gfCNCPoint4[15652] = {X 437.5566, Y 8.7395, Z -5.5000, A 0.000, B 0.000, C 0.000 }
gfCNCPoint4[15653] = {X 439.1460, Y 8.3375, Z -5.5000, A 0.000, B 0.000, C 0.000 }
gfCNCPoint4[15654] = {X 441.2360, Y 8.0482, Z -5.5000, A 0.000, B 0.000, C 0.000 }
gfCNCPoint4[15655] = {X 443.3437, Y 7.9543, Z -5.5000, A 0.000, B 0.000, C 0.000 }
gfCNCPoint4[15656] = {X 444.0360, Y 7.9502, Z -5.5000, A 0.000, B 0.000, C 0.000 }
gfCNCPoint4[15657] = {X 459.4468, Y 7.9502, Z -5.5000, A 0.000, B 0.000, C 0.000 }
gfCNCPoint4[15658] = {X 460.3883, Y 8.0563, Z -5.5000, A 0.000, B 0.000, C 0.000 }
gfCNCPoint4[15659] = {X 461.2826, Y 8.3693, Z -5.5000, A 0.000, B 0.000, C 0.000 }
gfCNCPoint4[15660] = {X 462.0849, Y 8.8733, Z -5.5000, A 0.000, B 0.000, C 0.000 }
gfCNCPoint4[15661] = {X 462.7548, Y 9.5433, Z -5.5000, A 0.000, B 0.000, C 0.000 }
gfCNCPoint4[15662] = {X 463.2589, Y 10.3456, Z -5.5000, A 0.000, B 0.000, C 0.000 }
gfCNCPoint4[15663] = {X 463.5719, Y 11.2399, Z -5.5000, A 0.000, B 0.000, C 0.000 }
gfCNCPoint4[15664] = {X 463.6779, Y 12.1814, Z -5.5000, A 0.000, B 0.000, C 0.000 }
gfCNCPoint4[15665] = {X 463.6779, Y 12.9782, Z -5.5000, A 0.000, B 0.000, C 0.000 }
gfCNCPoint4[15666] = {X 463.5765, Y 13.8997, Z -5.5000, A 0.000, B 0.000, C 0.000 }
gfCNCPoint4[15667] = {X 463.2771, Y 14.7771, Z -5.5000, A 0.000, B 0.000, C 0.000 }
gfCNCPoint4[15668] = {X 462.7943, Y 15.5685, Z -5.5000, A 0.000, B 0.000, C 0.000 }
gfCNCPoint4[15669] = {X 462.1509, Y 16.2360, Z -5.5000, A 0.000, B 0.000, C 0.000 }
gfCNCPoint4[15670] = {X 462.1511, Y 28.5935, Z -5.5000, A 0.000, B 0.000, C 0.000 }
gfCNCPoint4[15671] = {X 466.1511, Y 28.5934, Z -5.5000, A 0.000, B 0.000, C 0.000 }
gfCNCPoint4[15672] = {X 462.0711, Y 28.5935, Z -5.5000, A 0.000, B 0.000, C 0.000 }
gfCNCPoint4[15673] = {X 462.0714, Y 40.9895, Z -5.5000, A 0.000, B 0.000, C 0.000 }
gfCNCPoint4[15674] = {X 462.1372, Y 41.0434, Z -5.5000, A 0.000, B 0.000, C 0.000 }
gfCNCPoint4[15675] = {X 462.7480, Y 41.6890, Z -5.5000, A 0.000, B 0.000, C 0.000 }
gfCNCPoint4[15676] = {X 463.2076, Y 42.4496, Z -5.5000, A 0.000, B 0.000, C 0.000 }
gfCNCPoint4[15677] = {X 463.4953, Y 43.2904, Z -5.5000, A 0.000, B 0.000, C 0.000 }
gfCNCPoint4[15678] = {X 463.5978, Y 44.1731, Z -5.5000, A 0.000, B 0.000, C 0.000 }
gfCNCPoint4[15679] = {X 463.5979, Y 45.0000, Z -5.5000, A 0.000, B 0.000, C 0.000 }
gfCNCPoint4[15680] = {X 463.4936, Y 45.9257, Z -5.5000, A 0.000, B 0.000, C 0.000 }
gfCNCPoint4[15681] = {X 463.1860, Y 46.8050, Z -5.5000, A 0.000, B 0.000, C 0.000 }
gfCNCPoint4[15682] = {X 462.6904, Y 47.5937, Z -5.5000, A 0.000, B 0.000, C 0.000 }
gfCNCPoint4[15683] = {X 462.0317, Y 48.2524, Z -5.5000, A 0.000, B 0.000, C 0.000 }
gfCNCPoint4[15684] = {X 461.2429, Y 48.7480, Z -5.5000, A 0.000, B 0.000, C 0.000 }
gfCNCPoint4[15685] = {X 460.3636, Y 49.0557, Z -5.5000, A 0.000, B 0.000, C 0.000 }
gfCNCPoint4[15686] = {X 459.4379, Y 49.1600, Z -5.5000, A 0.000, B 0.000, C 0.000 }
gfCNCPoint4[15687] = {X 452.9945, Y 49.1600, Z -5.5000, A 0.000, B 0.000, C 0.000 }
gfCNCPoint4[15688] = {X 452.0735, Y 49.0568, Z -5.5000, A 0.000, B 0.000, C 0.000 }
gfCNCPoint4[15689] = {X 451.1982, Y 48.7522, Z -5.5000, A 0.000, B 0.000, C 0.000 }
gfCNCPoint4[15690] = {X 450.4120, Y 48.2614, Z -5.5000, A 0.000, B 0.000, C 0.000 }
gfCNCPoint4[15691] = {X 449.7541, Y 47.6087, Z -5.5000, A 0.000, B 0.000, C 0.000 }
gfCNCPoint4[15692] = {X 449.2569, Y 46.8266, Z -5.5000, A 0.000, B 0.000, C 0.000 }
gfCNCPoint4[15693] = {X 448.9453, Y 45.9538, Z -5.5000, A 0.000, B 0.000, C 0.000 }
gfCNCPoint4[15694] = {X 448.8346, Y 45.0336, Z -5.5000, A 0.000, B 0.000, C 0.000 }
gfCNCPoint4[15695] = {X 448.8349, Y 44.1516, Z -5.5000, A 0.000, B 0.000, C 0.000 }
gfCNCPoint4[15696] = {X 448.9454, Y 43.2545, Z -5.5000, A 0.000, B 0.000, C 0.000 }
gfCNCPoint4[15697] = {X 449.2471, Y 42.4026, Z -5.5000, A 0.000, B 0.000, C 0.000 }
gfCNCPoint4[15698] = {X 449.7256, Y 41.6358, Z -5.5000, A 0.000, B 0.000, C 0.000 }
gfCNCPoint4[15699] = {X 450.3584, Y 40.9906, Z -5.5000, A 0.000, B 0.000, C 0.000 }
gfCNCPoint4[15700] = {X 450.3584, Y 34.3138, Z -5.5000, A 0.000, B 0.000, C 0.000 }
gfCNCPoint4[15701] = {X 447.3773, Y 34.3138, Z -5.5000, A 0.000, B 0.000, C 0.000 }
gfCNCPoint4[15702] = {X 443.0156, Y 42.8061, Z -5.5000, A 0.000, B 0.000, C 0.000 }
gfCNCPoint4[15703] = {X 443.0437, Y 42.8834, Z -5.5000, A 0.000, B 0.000, C 0.000 }
gfCNCPoint4[15704] = {X 443.2029, Y 43.5190, Z -5.5000, A 0.000, B 0.000, C 0.000 }
gfCNCPoint4[15705] = {X 443.2603, Y 44.1717, Z -5.5000, A 0.000, B 0.000, C 0.000 }
gfCNCPoint4[15706] = {X 443.2605, Y 45.0000, Z -5.5000, A 0.000, B 0.000, C 0.000 }
gfCNCPoint4[15707] = {X 443.1562, Y 45.9257, Z -5.5000, A 0.000, B 0.000, C 0.000 }
gfCNCPoint4[15708] = {X 442.8485, Y 46.8050, Z -5.5000, A 0.000, B 0.000, C 0.000 }
gfCNCPoint4[15709] = {X 442.3529, Y 47.5937, Z -5.5000, A 0.000, B 0.000, C 0.000 }
gfCNCPoint4[15710] = {X 441.6942, Y 48.2524, Z -5.5000, A 0.000, B 0.000, C 0.000 }
gfCNCPoint4[15711] = {X 440.9054, Y 48.7480, Z -5.5000, A 0.000, B 0.000, C 0.000 }
gfCNCPoint4[15712] = {X 440.0262, Y 49.0557, Z -5.5000, A 0.000, B 0.000, C 0.000 }
gfCNCPoint4[15713] = {X 439.1005, Y 49.1600, Z -5.5000, A 0.000, B 0.000, C 0.000 }
gfCNCPoint4[15714] = {X 432.5144, Y 49.1600, Z -5.5000, A 0.000, B 0.000, C 0.000 }
gfCNCPoint4[15715] = {X 431.5887, Y 49.0557, Z -5.5000, A 0.000, B 0.000, C 0.000 }
gfCNCPoint4[15716] = {X 430.7095, Y 48.7480, Z -5.5000, A 0.000, B 0.000, C 0.000 }
gfCNCPoint4[15717] = {X 429.9207, Y 48.2524, Z -5.5000, A 0.000, B 0.000, C 0.000 }
gfCNCPoint4[15718] = {X 429.2620, Y 47.5937, Z -5.5000, A 0.000, B 0.000, C 0.000 }
gfCNCPoint4[15719] = {X 428.7664, Y 46.8050, Z -5.5000, A 0.000, B 0.000, C 0.000 }
gfCNCPoint4[15720] = {X 428.4587, Y 45.9257, Z -5.5000, A 0.000, B 0.000, C 0.000 }
gfCNCPoint4[15721] = {X 428.3544, Y 45.0000, Z -5.5000, A 0.000, B 0.000, C 0.000 }
gfCNCPoint4[15722] = {X 428.3548, Y 44.1516, Z -5.5000, A 0.000, B 0.000, C 0.000 }
gfCNCPoint4[15723] = {X 428.4510, Y 43.3174, Z -5.5000, A 0.000, B 0.000, C 0.000 }
gfCNCPoint4[15724] = {X 428.7128, Y 42.5195, Z -5.5000, A 0.000, B 0.000, C 0.000 }
gfCNCPoint4[15725] = {X 429.1295, Y 41.7905, Z -5.5000, A 0.000, B 0.000, C 0.000 }
gfCNCPoint4[15726] = {X 429.6841, Y 41.1600, Z -5.5000, A 0.000, B 0.000, C 0.000 }
gfCNCPoint4[15727] = {X 430.3541, Y 40.6537, Z -5.5000, A 0.000, B 0.000, C 0.000 }
gfCNCPoint4[15728] = {X 431.1120, Y 40.2923, Z -5.5000, A 0.000, B 0.000, C 0.000 }
gfCNCPoint4[15729] = {X 435.1988, Y 32.2929, Z -5.5000, A 0.000, B 0.000, C 0.000 }
gfCNCPoint4[15730] = {X 433.9189, Y 31.4434, Z -5.5000, A 0.000, B 0.000, C 0.000 }
gfCNCPoint4[15731] = {X 432.7670, Y 30.4271, Z -5.5000, A 0.000, B 0.000, C 0.000 }
gfCNCPoint4[15732] = {X 431.7646, Y 29.2630, Z -5.5000, A 0.000, B 0.000, C 0.000 }
gfCNCPoint4[15733] = {X 430.9305, Y 27.9730, Z -5.5000, A 0.000, B 0.000, C 0.000 }
gfCNCPoint4[15734] = {X 430.2803, Y 26.5812, Z -5.5000, A 0.000, B 0.000, C 0.000 }
gfCNCPoint4[15735] = {X 429.8262, Y 25.1137, Z -5.5000, A 0.000, B 0.000, C 0.000 }
gfCNCPoint4[15736] = {X 429.5151, Y 23.4467, Z -5.5000, A 0.000, B 0.000, C 0.000 }
gfCNCPoint4[15737] = {X 429.3761, Y 21.7566, Z -5.5000, A 0.000, B 0.000, C 0.000 }
gfCNCPoint4[15738] = {X 429.4105, Y 20.0612, Z -5.5000, A 0.000, B 0.000, C 0.000 }
gfCNCPoint4[15739] = {X 429.6179, Y 18.3782, Z -5.5000, A 0.000, B 0.000, C 0.000 }
gfCNCPoint4[15740] = {X 429.9963, Y 16.7251, Z -5.5000, A 0.000, B 0.000, C 0.000 }
gfCNCPoint4[15741] = {X 430.5478, Y 15.1930, Z -5.5000, A 0.000, B 0.000, C 0.000 }
gfCNCPoint4[15742] = {X 431.3072, Y 13.7525, Z -5.5000, A 0.000, B 0.000, C 0.000 }
gfCNCPoint4[15743] = {X 432.2597, Y 12.4318, Z -5.5000, A 0.000, B 0.000, C 0.000 }
gfCNCPoint4[15744] = {X 433.3868, Y 11.2565, Z -5.5000, A 0.000, B 0.000, C 0.000 }
gfCNCPoint4[15745] = {X 434.6666, Y 10.2495, Z -5.5000, A 0.000, B 0.000, C 0.000 }
gfCNCPoint4[15746] = {X 436.0740, Y 9.4305, Z -5.5000, A 0.000, B 0.000, C 0.000 }
gfCNCPoint4[15747] = {X 437.5818, Y 8.8154, Z -5.5000, A 0.000, B 0.000, C 0.000 }
gfCNCPoint4[15748] = {X 439.1605, Y 8.4162, Z -5.5000, A 0.000, B 0.000, C 0.000 }
gfCNCPoint4[15749] = {X 441.2433, Y 8.1279, Z -5.5000, A 0.000, B 0.000, C 0.000 }
gfCNCPoint4[15750] = {X 443.3439, Y 8.0343, Z -5.5000, A 0.000, B 0.000, C 0.000 }
gfCNCPoint4[15751] = {X 444.0362, Y 8.0302, Z -5.5000, A 0.000, B 0.000, C 0.000 }
gfCNCPoint4[15752] = {X 459.4468, Y 8.0302, Z -5.5000, A 0.000, B 0.000, C 0.000 }
gfCNCPoint4[15753] = {X 460.3705, Y 8.1343, Z -5.5000, A 0.000, B 0.000, C 0.000 }
gfCNCPoint4[15754] = {X 461.2479, Y 8.4413, Z -5.5000, A 0.000, B 0.000, C 0.000 }
gfCNCPoint4[15755] = {X 462.0350, Y 8.9359, Z -5.5000, A 0.000, B 0.000, C 0.000 }
gfCNCPoint4[15756] = {X 462.6923, Y 9.5932, Z -5.5000, A 0.000, B 0.000, C 0.000 }
gfCNCPoint4[15757] = {X 463.1868, Y 10.3803, Z -5.5000, A 0.000, B 0.000, C 0.000 }
gfCNCPoint4[15758] = {X 463.4939, Y 11.2577, Z -5.5000, A 0.000, B 0.000, C 0.000 }
gfCNCPoint4[15759] = {X 463.5979, Y 12.1814, Z -5.5000, A 0.000, B 0.000, C 0.000 }
gfCNCPoint4[15760] = {X 463.5979, Y 12.9782, Z -5.5000, A 0.000, B 0.000, C 0.000 }
gfCNCPoint4[15761] = {X 463.5023, Y 13.8650, Z -5.5000, A 0.000, B 0.000, C 0.000 }
gfCNCPoint4[15762] = {X 463.2198, Y 14.7111, Z -5.5000, A 0.000, B 0.000, C 0.000 }
gfCNCPoint4[15763] = {X 462.7634, Y 15.4774, Z -5.5000, A 0.000, B 0.000, C 0.000 }
gfCNCPoint4[15764] = {X 462.1541, Y 16.1289, Z -5.5000, A 0.000, B 0.000, C 0.000 }
gfCNCPoint4[15765] = {X 462.0709, Y 16.1987, Z -5.5000, A 0.000, B 0.000, C 0.000 }
gfCNCPoint4[15766] = {X 462.0711, Y 28.5935, Z -5.5000, A 0.000, B 0.000, C 0.000 }
gfCNCPoint4[15767] = {X 466.0711, Y 28.5934, Z -5.5000, A 0.000, B 0.000, C 0.000 }
gfCNCPoint4[15768] = {X 461.9911, Y 28.5935, Z -5.5000, A 0.000, B 0.000, C 0.000 }
gfCNCPoint4[15769] = {X 461.9914, Y 41.0273, Z -5.5000, A 0.000, B 0.000, C 0.000 }
gfCNCPoint4[15770] = {X 462.0859, Y 41.1048, Z -5.5000, A 0.000, B 0.000, C 0.000 }
gfCNCPoint4[15771] = {X 462.6847, Y 41.7379, Z -5.5000, A 0.000, B 0.000, C 0.000 }
gfCNCPoint4[15772] = {X 463.1353, Y 42.4837, Z -5.5000, A 0.000, B 0.000, C 0.000 }
gfCNCPoint4[15773] = {X 463.4173, Y 43.3082, Z -5.5000, A 0.000, B 0.000, C 0.000 }
gfCNCPoint4[15774] = {X 463.5178, Y 44.1738, Z -5.5000, A 0.000, B 0.000, C 0.000 }
gfCNCPoint4[15775] = {X 463.5179, Y 45.0000, Z -5.5000, A 0.000, B 0.000, C 0.000 }
gfCNCPoint4[15776] = {X 463.4156, Y 45.9079, Z -5.5000, A 0.000, B 0.000, C 0.000 }
gfCNCPoint4[15777] = {X 463.1139, Y 46.7702, Z -5.5000, A 0.000, B 0.000, C 0.000 }
gfCNCPoint4[15778] = {X 462.6278, Y 47.5438, Z -5.5000, A 0.000, B 0.000, C 0.000 }
gfCNCPoint4[15779] = {X 461.9818, Y 48.1899, Z -5.5000, A 0.000, B 0.000, C 0.000 }
gfCNCPoint4[15780] = {X 461.2082, Y 48.6760, Z -5.5000, A 0.000, B 0.000, C 0.000 }
gfCNCPoint4[15781] = {X 460.3458, Y 48.9777, Z -5.5000, A 0.000, B 0.000, C 0.000 }
gfCNCPoint4[15782] = {X 459.4379, Y 49.0800, Z -5.5000, A 0.000, B 0.000, C 0.000 }
gfCNCPoint4[15783] = {X 452.9945, Y 49.0800, Z -5.5000, A 0.000, B 0.000, C 0.000 }
gfCNCPoint4[15784] = {X 452.0912, Y 48.9788, Z -5.5000, A 0.000, B 0.000, C 0.000 }
gfCNCPoint4[15785] = {X 451.2327, Y 48.6800, Z -5.5000, A 0.000, B 0.000, C 0.000 }
gfCNCPoint4[15786] = {X 450.4617, Y 48.1987, Z -5.5000, A 0.000, B 0.000, C 0.000 }
gfCNCPoint4[15787] = {X 449.8164, Y 47.5585, Z -5.5000, A 0.000, B 0.000, C 0.000 }
gfCNCPoint4[15788] = {X 449.3288, Y 46.7914, Z -5.5000, A 0.000, B 0.000, C 0.000 }
gfCNCPoint4[15789] = {X 449.0232, Y 45.9354, Z -5.5000, A 0.000, B 0.000, C 0.000 }
gfCNCPoint4[15790] = {X 448.9146, Y 45.0330, Z -5.5000, A 0.000, B 0.000, C 0.000 }
gfCNCPoint4[15791] = {X 448.9149, Y 44.1527, Z -5.5000, A 0.000, B 0.000, C 0.000 }
gfCNCPoint4[15792] = {X 449.0254, Y 43.2637, Z -5.5000, A 0.000, B 0.000, C 0.000 }
gfCNCPoint4[15793] = {X 449.3274, Y 42.4203, Z -5.5000, A 0.000, B 0.000, C 0.000 }
gfCNCPoint4[15794] = {X 449.8061, Y 41.6631, Z -5.5000, A 0.000, B 0.000, C 0.000 }
gfCNCPoint4[15795] = {X 450.4384, Y 41.0287, Z -5.5000, A 0.000, B 0.000, C 0.000 }
gfCNCPoint4[15796] = {X 450.4384, Y 34.2338, Z -5.5000, A 0.000, B 0.000, C 0.000 }
gfCNCPoint4[15797] = {X 447.3284, Y 34.2338, Z -5.5000, A 0.000, B 0.000, C 0.000 }
gfCNCPoint4[15798] = {X 442.9284, Y 42.8006, Z -5.5000, A 0.000, B 0.000, C 0.000 }
gfCNCPoint4[15799] = {X 442.9682, Y 42.9099, Z -5.5000, A 0.000, B 0.000, C 0.000 }
gfCNCPoint4[15800] = {X 443.1241, Y 43.5328, Z -5.5000, A 0.000, B 0.000, C 0.000 }
gfCNCPoint4[15801] = {X 443.1803, Y 44.1725, Z -5.5000, A 0.000, B 0.000, C 0.000 }
gfCNCPoint4[15802] = {X 443.1805, Y 45.0000, Z -5.5000, A 0.000, B 0.000, C 0.000 }
gfCNCPoint4[15803] = {X 443.0782, Y 45.9079, Z -5.5000, A 0.000, B 0.000, C 0.000 }
gfCNCPoint4[15804] = {X 442.7764, Y 46.7702, Z -5.5000, A 0.000, B 0.000, C 0.000 }
gfCNCPoint4[15805] = {X 442.2903, Y 47.5438, Z -5.5000, A 0.000, B 0.000, C 0.000 }
gfCNCPoint4[15806] = {X 441.6443, Y 48.1899, Z -5.5000, A 0.000, B 0.000, C 0.000 }
gfCNCPoint4[15807] = {X 440.8707, Y 48.6760, Z -5.5000, A 0.000, B 0.000, C 0.000 }
gfCNCPoint4[15808] = {X 440.0084, Y 48.9777, Z -5.5000, A 0.000, B 0.000, C 0.000 }
gfCNCPoint4[15809] = {X 439.1005, Y 49.0800, Z -5.5000, A 0.000, B 0.000, C 0.000 }
gfCNCPoint4[15810] = {X 432.5144, Y 49.0800, Z -5.5000, A 0.000, B 0.000, C 0.000 }
gfCNCPoint4[15811] = {X 431.6065, Y 48.9777, Z -5.5000, A 0.000, B 0.000, C 0.000 }
gfCNCPoint4[15812] = {X 430.7442, Y 48.6760, Z -5.5000, A 0.000, B 0.000, C 0.000 }
gfCNCPoint4[15813] = {X 429.9706, Y 48.1899, Z -5.5000, A 0.000, B 0.000, C 0.000 }
gfCNCPoint4[15814] = {X 429.3245, Y 47.5438, Z -5.5000, A 0.000, B 0.000, C 0.000 }
gfCNCPoint4[15815] = {X 428.8385, Y 46.7702, Z -5.5000, A 0.000, B 0.000, C 0.000 }
gfCNCPoint4[15816] = {X 428.5367, Y 45.9079, Z -5.5000, A 0.000, B 0.000, C 0.000 }
gfCNCPoint4[15817] = {X 428.4344, Y 45.0000, Z -5.5000, A 0.000, B 0.000, C 0.000 }
gfCNCPoint4[15818] = {X 428.4348, Y 44.1527, Z -5.5000, A 0.000, B 0.000, C 0.000 }
gfCNCPoint4[15819] = {X 428.5303, Y 43.3294, Z -5.5000, A 0.000, B 0.000, C 0.000 }
gfCNCPoint4[15820] = {X 428.7902, Y 42.5424, Z -5.5000, A 0.000, B 0.000, C 0.000 }
gfCNCPoint4[15821] = {X 429.2038, Y 41.8242, Z -5.5000, A 0.000, B 0.000, C 0.000 }
gfCNCPoint4[15822] = {X 429.7540, Y 41.2044, Z -5.5000, A 0.000, B 0.000, C 0.000 }
gfCNCPoint4[15823] = {X 430.4181, Y 40.7085, Z -5.5000, A 0.000, B 0.000, C 0.000 }
gfCNCPoint4[15824] = {X 431.1687, Y 40.3571, Z -5.5000, A 0.000, B 0.000, C 0.000 }
gfCNCPoint4[15825] = {X 435.3049, Y 32.2610, Z -5.5000, A 0.000, B 0.000, C 0.000 }
gfCNCPoint4[15826] = {X 434.0182, Y 31.4185, Z -5.5000, A 0.000, B 0.000, C 0.000 }
gfCNCPoint4[15827] = {X 432.8597, Y 30.4069, Z -5.5000, A 0.000, B 0.000, C 0.000 }
gfCNCPoint4[15828] = {X 431.8515, Y 29.2455, Z -5.5000, A 0.000, B 0.000, C 0.000 }
gfCNCPoint4[15829] = {X 431.0128, Y 27.9564, Z -5.5000, A 0.000, B 0.000, C 0.000 }
gfCNCPoint4[15830] = {X 430.3595, Y 26.5641, Z -5.5000, A 0.000, B 0.000, C 0.000 }
gfCNCPoint4[15831] = {X 429.9040, Y 25.0951, Z -5.5000, A 0.000, B 0.000, C 0.000 }
gfCNCPoint4[15832] = {X 429.5944, Y 23.4361, Z -5.5000, A 0.000, B 0.000, C 0.000 }
gfCNCPoint4[15833] = {X 429.4560, Y 21.7542, Z -5.5000, A 0.000, B 0.000, C 0.000 }
gfCNCPoint4[15834] = {X 429.4902, Y 20.0670, Z -5.5000, A 0.000, B 0.000, C 0.000 }
gfCNCPoint4[15835] = {X 429.6967, Y 18.3920, Z -5.5000, A 0.000, B 0.000, C 0.000 }
gfCNCPoint4[15836] = {X 430.0732, Y 16.7470, Z -5.5000, A 0.000, B 0.000, C 0.000 }
gfCNCPoint4[15837] = {X 430.6210, Y 15.2253, Z -5.5000, A 0.000, B 0.000, C 0.000 }
gfCNCPoint4[15838] = {X 431.3752, Y 13.7946, Z -5.5000, A 0.000, B 0.000, C 0.000 }
gfCNCPoint4[15839] = {X 432.3212, Y 12.4829, Z -5.5000, A 0.000, B 0.000, C 0.000 }
gfCNCPoint4[15840] = {X 433.4406, Y 11.3157, Z -5.5000, A 0.000, B 0.000, C 0.000 }
gfCNCPoint4[15841] = {X 434.7116, Y 10.3156, Z -5.5000, A 0.000, B 0.000, C 0.000 }
gfCNCPoint4[15842] = {X 436.1095, Y 9.5022, Z -5.5000, A 0.000, B 0.000, C 0.000 }
gfCNCPoint4[15843] = {X 437.6070, Y 8.8914, Z -5.5000, A 0.000, B 0.000, C 0.000 }
gfCNCPoint4[15844] = {X 439.1749, Y 8.4949, Z -5.5000, A 0.000, B 0.000, C 0.000 }
gfCNCPoint4[15845] = {X 441.2506, Y 8.2075, Z -5.5000, A 0.000, B 0.000, C 0.000 }
gfCNCPoint4[15846] = {X 443.3440, Y 8.1143, Z -5.5000, A 0.000, B 0.000, C 0.000 }
gfCNCPoint4[15847] = {X 444.0364, Y 8.1102, Z -5.5000, A 0.000, B 0.000, C 0.000 }
gfCNCPoint4[15848] = {X 459.4468, Y 8.1102, Z -5.5000, A 0.000, B 0.000, C 0.000 }
gfCNCPoint4[15849] = {X 460.3527, Y 8.2123, Z -5.5000, A 0.000, B 0.000, C 0.000 }
gfCNCPoint4[15850] = {X 461.2132, Y 8.5134, Z -5.5000, A 0.000, B 0.000, C 0.000 }
gfCNCPoint4[15851] = {X 461.9851, Y 8.9984, Z -5.5000, A 0.000, B 0.000, C 0.000 }
gfCNCPoint4[15852] = {X 462.6297, Y 9.6431, Z -5.5000, A 0.000, B 0.000, C 0.000 }
gfCNCPoint4[15853] = {X 463.1148, Y 10.4150, Z -5.5000, A 0.000, B 0.000, C 0.000 }
gfCNCPoint4[15854] = {X 463.4159, Y 11.2755, Z -5.5000, A 0.000, B 0.000, C 0.000 }
gfCNCPoint4[15855] = {X 463.5179, Y 12.1814, Z -5.5000, A 0.000, B 0.000, C 0.000 }
gfCNCPoint4[15856] = {X 463.5179, Y 12.9781, Z -5.5000, A 0.000, B 0.000, C 0.000 }
gfCNCPoint4[15857] = {X 463.4241, Y 13.8479, Z -5.5000, A 0.000, B 0.000, C 0.000 }
gfCNCPoint4[15858] = {X 463.1470, Y 14.6777, Z -5.5000, A 0.000, B 0.000, C 0.000 }
gfCNCPoint4[15859] = {X 462.6994, Y 15.4294, Z -5.5000, A 0.000, B 0.000, C 0.000 }
gfCNCPoint4[15860] = {X 462.1019, Y 16.0683, Z -5.5000, A 0.000, B 0.000, C 0.000 }
gfCNCPoint4[15861] = {X 462.0444, Y 16.1170, Z -5.5000, A 0.000, B 0.000, C 0.000 }
gfCNCPoint4[15862] = {X 461.9860, Y 16.1646, Z -5.5000, A 0.000, B 0.000, C 0.000 }
gfCNCPoint4[15863] = {X 461.9909, Y 16.1987, Z -5.5000, A 0.000, B 0.000, C 0.000 }
gfCNCPoint4[15864] = {X 461.9911, Y 28.5935, Z -5.5000, A 0.000, B 0.000, C 0.000 }
gfCNCPoint4[15865] = {X 465.9911, Y 28.5934, Z -5.5000, A 0.000, B 0.000, C 0.000 }
gfCNCPoint4[15866] = {X 465.9911, Y 28.5933, Z -5.5000, A 0.000, B 0.000, C 0.000 }
gfCNCPoint4[15867] = {X 461.9108, Y 28.5935, Z -5.5000, A 0.000, B 0.000, C 0.000 }
gfCNCPoint4[15868] = {X 461.9114, Y 41.0652, Z -5.5000, A 0.000, B 0.000, C 0.000 }
gfCNCPoint4[15869] = {X 462.0501, Y 41.1795, Z -5.5000, A 0.000, B 0.000, C 0.000 }
gfCNCPoint4[15870] = {X 462.6358, Y 41.8059, Z -5.5000, A 0.000, B 0.000, C 0.000 }
gfCNCPoint4[15871] = {X 463.0745, Y 42.5428, Z -5.5000, A 0.000, B 0.000, C 0.000 }
gfCNCPoint4[15872] = {X 463.3460, Y 43.3562, Z -5.5000, A 0.000, B 0.000, C 0.000 }
gfCNCPoint4[15873] = {X 463.4379, Y 44.2089, Z -5.5000, A 0.000, B 0.000, C 0.000 }
gfCNCPoint4[15874] = {X 463.4379, Y 45.0000, Z -5.5000, A 0.000, B 0.000, C 0.000 }
gfCNCPoint4[15875] = {X 463.3377, Y 45.8901, Z -5.5000, A 0.000, B 0.000, C 0.000 }
gfCNCPoint4[15876] = {X 463.0418, Y 46.7355, Z -5.5000, A 0.000, B 0.000, C 0.000 }
gfCNCPoint4[15877] = {X 462.5653, Y 47.4940, Z -5.5000, A 0.000, B 0.000, C 0.000 }
gfCNCPoint4[15878] = {X 461.9319, Y 48.1273, Z -5.5000, A 0.000, B 0.000, C 0.000 }
gfCNCPoint4[15879] = {X 461.1735, Y 48.6039, Z -5.5000, A 0.000, B 0.000, C 0.000 }
gfCNCPoint4[15880] = {X 460.3280, Y 48.8997, Z -5.5000, A 0.000, B 0.000, C 0.000 }
gfCNCPoint4[15881] = {X 459.4379, Y 49.0000, Z -5.5000, A 0.000, B 0.000, C 0.000 }
gfCNCPoint4[15882] = {X 452.9945, Y 49.0000, Z -5.5000, A 0.000, B 0.000, C 0.000 }
gfCNCPoint4[15883] = {X 452.1044, Y 48.8997, Z -5.5000, A 0.000, B 0.000, C 0.000 }
gfCNCPoint4[15884] = {X 451.2589, Y 48.6039, Z -5.5000, A 0.000, B 0.000, C 0.000 }
gfCNCPoint4[15885] = {X 450.5005, Y 48.1273, Z -5.5000, A 0.000, B 0.000, C 0.000 }
gfCNCPoint4[15886] = {X 449.8671, Y 47.4939, Z -5.5000, A 0.000, B 0.000, C 0.000 }
gfCNCPoint4[15887] = {X 449.3906, Y 46.7355, Z -5.5000, A 0.000, B 0.000, C 0.000 }
gfCNCPoint4[15888] = {X 449.0948, Y 45.8901, Z -5.5000, A 0.000, B 0.000, C 0.000 }
gfCNCPoint4[15889] = {X 448.9945, Y 45.0000, Z -5.5000, A 0.000, B 0.000, C 0.000 }
gfCNCPoint4[15890] = {X 448.9949, Y 44.1538, Z -5.5000, A 0.000, B 0.000, C 0.000 }
gfCNCPoint4[15891] = {X 449.1055, Y 43.2730, Z -5.5000, A 0.000, B 0.000, C 0.000 }
gfCNCPoint4[15892] = {X 449.4077, Y 42.4382, Z -5.5000, A 0.000, B 0.000, C 0.000 }
gfCNCPoint4[15893] = {X 449.8865, Y 41.6907, Z -5.5000, A 0.000, B 0.000, C 0.000 }
gfCNCPoint4[15894] = {X 450.5184, Y 41.0672, Z -5.5000, A 0.000, B 0.000, C 0.000 }
gfCNCPoint4[15895] = {X 450.5184, Y 34.1538, Z -5.5000, A 0.000, B 0.000, C 0.000 }
gfCNCPoint4[15896] = {X 447.5238, Y 34.1538, Z -5.5000, A 0.000, B 0.000, C 0.000 }
gfCNCPoint4[15897] = {X 447.2797, Y 34.1535, Z -5.5000, A 0.000, B 0.000, C 0.000 }
gfCNCPoint4[15898] = {X 442.8413, Y 42.7952, Z -5.5000, A 0.000, B 0.000, C 0.000 }
gfCNCPoint4[15899] = {X 442.8970, Y 42.9491, Z -5.5000, A 0.000, B 0.000, C 0.000 }
gfCNCPoint4[15900] = {X 443.0493, Y 43.5708, Z -5.5000, A 0.000, B 0.000, C 0.000 }
gfCNCPoint4[15901] = {X 443.1005, Y 44.2089, Z -5.5000, A 0.000, B 0.000, C 0.000 }
gfCNCPoint4[15902] = {X 443.1005, Y 45.0000, Z -5.5000, A 0.000, B 0.000, C 0.000 }
gfCNCPoint4[15903] = {X 443.0002, Y 45.8901, Z -5.5000, A 0.000, B 0.000, C 0.000 }
gfCNCPoint4[15904] = {X 442.7043, Y 46.7355, Z -5.5000, A 0.000, B 0.000, C 0.000 }
gfCNCPoint4[15905] = {X 442.2278, Y 47.4940, Z -5.5000, A 0.000, B 0.000, C 0.000 }
gfCNCPoint4[15906] = {X 441.5944, Y 48.1273, Z -5.5000, A 0.000, B 0.000, C 0.000 }
gfCNCPoint4[15907] = {X 440.8360, Y 48.6039, Z -5.5000, A 0.000, B 0.000, C 0.000 }
gfCNCPoint4[15908] = {X 439.9906, Y 48.8997, Z -5.5000, A 0.000, B 0.000, C 0.000 }
gfCNCPoint4[15909] = {X 439.1005, Y 49.0000, Z -5.5000, A 0.000, B 0.000, C 0.000 }
gfCNCPoint4[15910] = {X 432.5144, Y 49.0000, Z -5.5000, A 0.000, B 0.000, C 0.000 }
gfCNCPoint4[15911] = {X 431.6243, Y 48.8997, Z -5.5000, A 0.000, B 0.000, C 0.000 }
gfCNCPoint4[15912] = {X 430.7789, Y 48.6039, Z -5.5000, A 0.000, B 0.000, C 0.000 }
gfCNCPoint4[15913] = {X 430.0204, Y 48.1273, Z -5.5000, A 0.000, B 0.000, C 0.000 }
gfCNCPoint4[15914] = {X 429.3871, Y 47.4940, Z -5.5000, A 0.000, B 0.000, C 0.000 }
gfCNCPoint4[15915] = {X 428.9105, Y 46.7355, Z -5.5000, A 0.000, B 0.000, C 0.000 }
gfCNCPoint4[15916] = {X 428.6147, Y 45.8901, Z -5.5000, A 0.000, B 0.000, C 0.000 }
gfCNCPoint4[15917] = {X 428.5144, Y 45.0000, Z -5.5000, A 0.000, B 0.000, C 0.000 }
gfCNCPoint4[15918] = {X 428.5148, Y 44.1538, Z -5.5000, A 0.000, B 0.000, C 0.000 }
gfCNCPoint4[15919] = {X 428.6096, Y 43.3414, Z -5.5000, A 0.000, B 0.000, C 0.000 }
gfCNCPoint4[15920] = {X 428.8676, Y 42.5654, Z -5.5000, A 0.000, B 0.000, C 0.000 }
gfCNCPoint4[15921] = {X 429.2781, Y 41.8580, Z -5.5000, A 0.000, B 0.000, C 0.000 }
gfCNCPoint4[15922] = {X 429.8239, Y 41.2489, Z -5.5000, A 0.000, B 0.000, C 0.000 }
gfCNCPoint4[15923] = {X 430.4821, Y 40.7635, Z -5.5000, A 0.000, B 0.000, C 0.000 }
gfCNCPoint4[15924] = {X 431.2253, Y 40.4222, Z -5.5000, A 0.000, B 0.000, C 0.000 }
gfCNCPoint4[15925] = {X 435.4113, Y 32.2286, Z -5.5000, A 0.000, B 0.000, C 0.000 }
gfCNCPoint4[15926] = {X 434.1177, Y 31.3934, Z -5.5000, A 0.000, B 0.000, C 0.000 }
gfCNCPoint4[15927] = {X 432.9527, Y 30.3867, Z -5.5000, A 0.000, B 0.000, C 0.000 }
gfCNCPoint4[15928] = {X 431.9386, Y 29.2280, Z -5.5000, A 0.000, B 0.000, C 0.000 }
gfCNCPoint4[15929] = {X 431.0951, Y 27.9398, Z -5.5000, A 0.000, B 0.000, C 0.000 }
gfCNCPoint4[15930] = {X 430.4386, Y 26.5470, Z -5.5000, A 0.000, B 0.000, C 0.000 }
gfCNCPoint4[15931] = {X 429.9818, Y 25.0766, Z -5.5000, A 0.000, B 0.000, C 0.000 }
gfCNCPoint4[15932] = {X 429.6737, Y 23.4256, Z -5.5000, A 0.000, B 0.000, C 0.000 }
gfCNCPoint4[15933] = {X 429.5360, Y 21.7518, Z -5.5000, A 0.000, B 0.000, C 0.000 }
gfCNCPoint4[15934] = {X 429.5700, Y 20.0727, Z -5.5000, A 0.000, B 0.000, C 0.000 }
gfCNCPoint4[15935] = {X 429.7755, Y 18.4059, Z -5.5000, A 0.000, B 0.000, C 0.000 }
gfCNCPoint4[15936] = {X 430.1502, Y 16.7687, Z -5.5000, A 0.000, B 0.000, C 0.000 }
gfCNCPoint4[15937] = {X 430.6942, Y 15.2575, Z -5.5000, A 0.000, B 0.000, C 0.000 }
gfCNCPoint4[15938] = {X 431.4432, Y 13.8367, Z -5.5000, A 0.000, B 0.000, C 0.000 }
gfCNCPoint4[15939] = {X 432.3827, Y 12.5340, Z -5.5000, A 0.000, B 0.000, C 0.000 }
gfCNCPoint4[15940] = {X 433.4945, Y 11.3748, Z -5.5000, A 0.000, B 0.000, C 0.000 }
gfCNCPoint4[15941] = {X 434.7567, Y 10.3817, Z -5.5000, A 0.000, B 0.000, C 0.000 }
gfCNCPoint4[15942] = {X 436.1450, Y 9.5739, Z -5.5000, A 0.000, B 0.000, C 0.000 }
gfCNCPoint4[15943] = {X 437.6321, Y 8.9673, Z -5.5000, A 0.000, B 0.000, C 0.000 }
gfCNCPoint4[15944] = {X 439.1893, Y 8.5736, Z -5.5000, A 0.000, B 0.000, C 0.000 }
gfCNCPoint4[15945] = {X 441.2579, Y 8.2872, Z -5.5000, A 0.000, B 0.000, C 0.000 }
gfCNCPoint4[15946] = {X 443.3442, Y 8.1943, Z -5.5000, A 0.000, B 0.000, C 0.000 }
gfCNCPoint4[15947] = {X 444.0367, Y 8.1902, Z -5.5000, A 0.000, B 0.000, C 0.000 }
gfCNCPoint4[15948] = {X 459.4468, Y 8.1902, Z -5.5000, A 0.000, B 0.000, C 0.000 }
gfCNCPoint4[15949] = {X 460.3349, Y 8.2903, Z -5.5000, A 0.000, B 0.000, C 0.000 }
gfCNCPoint4[15950] = {X 461.1785, Y 8.5855, Z -5.5000, A 0.000, B 0.000, C 0.000 }
gfCNCPoint4[15951] = {X 461.9352, Y 9.0610, Z -5.5000, A 0.000, B 0.000, C 0.000 }
gfCNCPoint4[15952] = {X 462.5672, Y 9.6930, Z -5.5000, A 0.000, B 0.000, C 0.000 }
gfCNCPoint4[15953] = {X 463.0427, Y 10.4497, Z -5.5000, A 0.000, B 0.000, C 0.000 }
gfCNCPoint4[15954] = {X 463.3379, Y 11.2933, Z -5.5000, A 0.000, B 0.000, C 0.000 }
gfCNCPoint4[15955] = {X 463.4379, Y 12.1814, Z -5.5000, A 0.000, B 0.000, C 0.000 }
gfCNCPoint4[15956] = {X 463.4378, Y 13.0163, Z -5.5000, A 0.000, B 0.000, C 0.000 }
gfCNCPoint4[15957] = {X 463.3398, Y 13.8588, Z -5.5000, A 0.000, B 0.000, C 0.000 }
gfCNCPoint4[15958] = {X 463.0663, Y 14.6617, Z -5.5000, A 0.000, B 0.000, C 0.000 }
gfCNCPoint4[15959] = {X 462.6297, Y 15.3889, Z -5.5000, A 0.000, B 0.000, C 0.000 }
gfCNCPoint4[15960] = {X 462.0496, Y 16.0077, Z -5.5000, A 0.000, B 0.000, C 0.000 }
gfCNCPoint4[15961] = {X 461.9727, Y 16.0724, Z -5.5000, A 0.000, B 0.000, C 0.000 }
gfCNCPoint4[15962] = {X 461.8942, Y 16.1351, Z -5.5000, A 0.000, B 0.000, C 0.000 }
gfCNCPoint4[15963] = {X 461.9109, Y 16.1931, Z -5.5000, A 0.000, B 0.000, C 0.000 }
gfCNCPoint4[15964] = {X 461.9103, Y 16.7687, Z -5.5000, A 0.000, B 0.000, C 0.000 }
gfCNCPoint4[15965] = {X 461.9108, Y 28.5935, Z -5.5000, A 0.000, B 0.000, C 0.000 }
gfCNCPoint4[15966] = {X 465.9911, Y 28.5933, Z -5.5000, A 0.000, B 0.000, C 0.000 }
gfCNCPoint4[15967] = {X 465.9911, Y 28.5933, Z -2.5000, A 0.000, B 0.000, C 0.000 }
gfCNCPoint4[15968] = {X 465.9911, Y 28.5933, Z 11.0000, A 0.000, B 0.000, C 0.000 }
gfCNCPoint4[15969] = {X 492.3835, Y 3.7902, Z 11.0000, A 0.000, B 0.000, C 0.000 }
gfCNCPoint4[15970] = {X 492.3835, Y 3.7902, Z -2.5000, A 0.000, B 0.000, C 0.000 }
gfCNCPoint4[15971] = {X 492.3835, Y 3.7902, Z -5.5000, A 0.000, B 0.000, C 0.000 }
gfCNCPoint4[15972] = {X 492.3835, Y 7.8702, Z -5.5000, A 0.000, B 0.000, C 0.000 }
gfCNCPoint4[15973] = {X 502.2066, Y 7.8702, Z -5.5000, A 0.000, B 0.000, C 0.000 }
gfCNCPoint4[15974] = {X 502.7395, Y 7.8744, Z -5.5000, A 0.000, B 0.000, C 0.000 }
gfCNCPoint4[15975] = {X 503.6914, Y 7.9886, Z -5.5000, A 0.000, B 0.000, C 0.000 }
gfCNCPoint4[15976] = {X 504.5943, Y 8.3108, Z -5.5000, A 0.000, B 0.000, C 0.000 }
gfCNCPoint4[15977] = {X 505.4035, Y 8.8250, Z -5.5000, A 0.000, B 0.000, C 0.000 }
gfCNCPoint4[15978] = {X 506.0788, Y 9.5055, Z -5.5000, A 0.000, B 0.000, C 0.000 }
gfCNCPoint4[15979] = {X 506.5866, Y 10.3187, Z -5.5000, A 0.000, B 0.000, C 0.000 }
gfCNCPoint4[15980] = {X 506.9017, Y 11.2241, Z -5.5000, A 0.000, B 0.000, C 0.000 }
gfCNCPoint4[15981] = {X 507.0085, Y 12.1769, Z -5.5000, A 0.000, B 0.000, C 0.000 }
gfCNCPoint4[15982] = {X 507.0085, Y 12.9782, Z -5.5000, A 0.000, B 0.000, C 0.000 }
gfCNCPoint4[15983] = {X 506.9072, Y 13.9080, Z -5.5000, A 0.000, B 0.000, C 0.000 }
gfCNCPoint4[15984] = {X 506.6082, Y 14.7942, Z -5.5000, A 0.000, B 0.000, C 0.000 }
gfCNCPoint4[15985] = {X 506.1254, Y 15.5953, Z -5.5000, A 0.000, B 0.000, C 0.000 }
gfCNCPoint4[15986] = {X 505.4815, Y 16.2737, Z -5.5000, A 0.000, B 0.000, C 0.000 }
gfCNCPoint4[15987] = {X 505.4814, Y 40.9131, Z -5.5000, A 0.000, B 0.000, C 0.000 }
gfCNCPoint4[15988] = {X 506.1197, Y 41.5840, Z -5.5000, A 0.000, B 0.000, C 0.000 }
gfCNCPoint4[15989] = {X 506.6003, Y 42.3756, Z -5.5000, A 0.000, B 0.000, C 0.000 }
gfCNCPoint4[15990] = {X 506.9011, Y 43.2515, Z -5.5000, A 0.000, B 0.000, C 0.000 }
gfCNCPoint4[15991] = {X 507.0083, Y 44.1713, Z -5.5000, A 0.000, B 0.000, C 0.000 }
gfCNCPoint4[15992] = {X 507.0085, Y 45.0000, Z -5.5000, A 0.000, B 0.000, C 0.000 }
gfCNCPoint4[15993] = {X 506.9002, Y 45.9613, Z -5.5000, A 0.000, B 0.000, C 0.000 }
gfCNCPoint4[15994] = {X 506.5807, Y 46.8744, Z -5.5000, A 0.000, B 0.000, C 0.000 }
gfCNCPoint4[15995] = {X 506.0660, Y 47.6935, Z -5.5000, A 0.000, B 0.000, C 0.000 }
gfCNCPoint4[15996] = {X 505.3820, Y 48.3775, Z -5.5000, A 0.000, B 0.000, C 0.000 }
gfCNCPoint4[15997] = {X 504.5629, Y 48.8922, Z -5.5000, A 0.000, B 0.000, C 0.000 }
gfCNCPoint4[15998] = {X 503.6498, Y 49.2117, Z -5.5000, A 0.000, B 0.000, C 0.000 }
gfCNCPoint4[15999] = {X 502.6885, Y 49.3200, Z -5.5000, A 0.000, B 0.000, C 0.000 }
gfCNCPoint4[16000] = {X 496.2450, Y 49.3200, Z -5.5000, A 0.000, B 0.000, C 0.000 }
gfCNCPoint4[16001] = {X 495.2885, Y 49.2128, Z -5.5000, A 0.000, B 0.000, C 0.000 }
gfCNCPoint4[16002] = {X 494.3794, Y 48.8964, Z -5.5000, A 0.000, B 0.000, C 0.000 }
gfCNCPoint4[16003] = {X 493.5630, Y 48.3866, Z -5.5000, A 0.000, B 0.000, C 0.000 }
gfCNCPoint4[16004] = {X 492.8797, Y 47.7087, Z -5.5000, A 0.000, B 0.000, C 0.000 }
gfCNCPoint4[16005] = {X 492.3635, Y 46.8963, Z -5.5000, A 0.000, B 0.000, C 0.000 }
gfCNCPoint4[16006] = {X 492.0399, Y 45.9898, Z -5.5000, A 0.000, B 0.000, C 0.000 }
gfCNCPoint4[16007] = {X 491.9252, Y 45.0341, Z -5.5000, A 0.000, B 0.000, C 0.000 }
gfCNCPoint4[16008] = {X 491.9254, Y 44.1494, Z -5.5000, A 0.000, B 0.000, C 0.000 }
gfCNCPoint4[16009] = {X 492.0359, Y 43.2364, Z -5.5000, A 0.000, B 0.000, C 0.000 }
gfCNCPoint4[16010] = {X 492.3371, Y 42.3675, Z -5.5000, A 0.000, B 0.000, C 0.000 }
gfCNCPoint4[16011] = {X 492.8153, Y 41.5821, Z -5.5000, A 0.000, B 0.000, C 0.000 }
gfCNCPoint4[16012] = {X 493.4490, Y 40.9157, Z -5.5000, A 0.000, B 0.000, C 0.000 }
gfCNCPoint4[16013] = {X 493.4490, Y 34.4738, Z -5.5000, A 0.000, B 0.000, C 0.000 }
gfCNCPoint4[16014] = {X 490.7248, Y 34.4738, Z -5.5000, A 0.000, B 0.000, C 0.000 }
gfCNCPoint4[16015] = {X 486.4404, Y 42.8174, Z -5.5000, A 0.000, B 0.000, C 0.000 }
gfCNCPoint4[16016] = {X 486.4451, Y 42.8302, Z -5.5000, A 0.000, B 0.000, C 0.000 }
gfCNCPoint4[16017] = {X 486.6110, Y 43.4911, Z -5.5000, A 0.000, B 0.000, C 0.000 }
gfCNCPoint4[16018] = {X 486.6708, Y 44.1699, Z -5.5000, A 0.000, B 0.000, C 0.000 }
gfCNCPoint4[16019] = {X 486.6710, Y 45.0000, Z -5.5000, A 0.000, B 0.000, C 0.000 }
gfCNCPoint4[16020] = {X 486.5627, Y 45.9613, Z -5.5000, A 0.000, B 0.000, C 0.000 }
gfCNCPoint4[16021] = {X 486.2432, Y 46.8744, Z -5.5000, A 0.000, B 0.000, C 0.000 }
gfCNCPoint4[16022] = {X 485.7285, Y 47.6935, Z -5.5000, A 0.000, B 0.000, C 0.000 }
gfCNCPoint4[16023] = {X 485.0445, Y 48.3775, Z -5.5000, A 0.000, B 0.000, C 0.000 }
gfCNCPoint4[16024] = {X 484.2254, Y 48.8922, Z -5.5000, A 0.000, B 0.000, C 0.000 }
gfCNCPoint4[16025] = {X 483.3123, Y 49.2117, Z -5.5000, A 0.000, B 0.000, C 0.000 }
gfCNCPoint4[16026] = {X 482.3510, Y 49.3200, Z -5.5000, A 0.000, B 0.000, C 0.000 }
gfCNCPoint4[16027] = {X 475.7650, Y 49.3200, Z -5.5000, A 0.000, B 0.000, C 0.000 }
gfCNCPoint4[16028] = {X 474.8037, Y 49.2117, Z -5.5000, A 0.000, B 0.000, C 0.000 }
gfCNCPoint4[16029] = {X 473.8906, Y 48.8922, Z -5.5000, A 0.000, B 0.000, C 0.000 }
gfCNCPoint4[16030] = {X 473.0715, Y 48.3775, Z -5.5000, A 0.000, B 0.000, C 0.000 }
gfCNCPoint4[16031] = {X 472.3875, Y 47.6935, Z -5.5000, A 0.000, B 0.000, C 0.000 }
gfCNCPoint4[16032] = {X 471.8728, Y 46.8744, Z -5.5000, A 0.000, B 0.000, C 0.000 }
gfCNCPoint4[16033] = {X 471.5533, Y 45.9614, Z -5.5000, A 0.000, B 0.000, C 0.000 }
gfCNCPoint4[16034] = {X 471.4450, Y 45.0001, Z -5.5000, A 0.000, B 0.000, C 0.000 }
gfCNCPoint4[16035] = {X 471.4454, Y 44.1494, Z -5.5000, A 0.000, B 0.000, C 0.000 }
gfCNCPoint4[16036] = {X 471.5430, Y 43.2935, Z -5.5000, A 0.000, B 0.000, C 0.000 }
gfCNCPoint4[16037] = {X 471.8086, Y 42.4740, Z -5.5000, A 0.000, B 0.000, C 0.000 }
gfCNCPoint4[16038] = {X 472.2314, Y 41.7236, Z -5.5000, A 0.000, B 0.000, C 0.000 }
gfCNCPoint4[16039] = {X 472.7947, Y 41.0719, Z -5.5000, A 0.000, B 0.000, C 0.000 }
gfCNCPoint4[16040] = {X 473.4762, Y 40.5449, Z -5.5000, A 0.000, B 0.000, C 0.000 }
gfCNCPoint4[16041] = {X 474.2486, Y 40.1637, Z -5.5000, A 0.000, B 0.000, C 0.000 }
gfCNCPoint4[16042] = {X 478.2330, Y 32.3647, Z -5.5000, A 0.000, B 0.000, C 0.000 }
gfCNCPoint4[16043] = {X 476.9689, Y 31.4976, Z -5.5000, A 0.000, B 0.000, C 0.000 }
gfCNCPoint4[16044] = {X 475.8320, Y 30.4694, Z -5.5000, A 0.000, B 0.000, C 0.000 }
gfCNCPoint4[16045] = {X 474.8426, Y 29.2987, Z -5.5000, A 0.000, B 0.000, C 0.000 }
gfCNCPoint4[16046] = {X 474.0183, Y 28.0063, Z -5.5000, A 0.000, B 0.000, C 0.000 }
gfCNCPoint4[16047] = {X 473.3739, Y 26.6154, Z -5.5000, A 0.000, B 0.000, C 0.000 }
gfCNCPoint4[16048] = {X 472.9211, Y 25.1509, Z -5.5000, A 0.000, B 0.000, C 0.000 }
gfCNCPoint4[16049] = {X 472.6070, Y 23.4679, Z -5.5000, A 0.000, B 0.000, C 0.000 }
gfCNCPoint4[16050] = {X 472.4666, Y 21.7615, Z -5.5000, A 0.000, B 0.000, C 0.000 }
gfCNCPoint4[16051] = {X 472.5013, Y 20.0497, Z -5.5000, A 0.000, B 0.000, C 0.000 }
gfCNCPoint4[16052] = {X 472.7108, Y 18.3505, Z -5.5000, A 0.000, B 0.000, C 0.000 }
gfCNCPoint4[16053] = {X 473.0928, Y 16.6815, Z -5.5000, A 0.000, B 0.000, C 0.000 }
gfCNCPoint4[16054] = {X 473.6356, Y 15.1666, Z -5.5000, A 0.000, B 0.000, C 0.000 }
gfCNCPoint4[16055] = {X 474.3790, Y 13.7394, Z -5.5000, A 0.000, B 0.000, C 0.000 }
gfCNCPoint4[16056] = {X 475.3091, Y 12.4262, Z -5.5000, A 0.000, B 0.000, C 0.000 }
gfCNCPoint4[16057] = {X 476.4088, Y 11.2514, Z -5.5000, A 0.000, B 0.000, C 0.000 }
gfCNCPoint4[16058] = {X 477.6578, Y 10.2367, Z -5.5000, A 0.000, B 0.000, C 0.000 }
gfCNCPoint4[16059] = {X 479.0329, Y 9.4008, Z -5.5000, A 0.000, B 0.000, C 0.000 }
gfCNCPoint4[16060] = {X 480.5087, Y 8.7593, Z -5.5000, A 0.000, B 0.000, C 0.000 }
gfCNCPoint4[16061] = {X 482.0579, Y 8.3239, Z -5.5000, A 0.000, B 0.000, C 0.000 }
gfCNCPoint4[16062] = {X 484.1552, Y 7.9971, Z -5.5000, A 0.000, B 0.000, C 0.000 }
gfCNCPoint4[16063] = {X 486.2747, Y 7.8824, Z -5.5000, A 0.000, B 0.000, C 0.000 }
gfCNCPoint4[16064] = {X 486.9679, Y 7.8702, Z -5.5000, A 0.000, B 0.000, C 0.000 }
gfCNCPoint4[16065] = {X 492.3835, Y 7.8702, Z -5.5000, A 0.000, B 0.000, C 0.000 }
gfCNCPoint4[16066] = {X 492.3835, Y 3.8702, Z -5.5000, A 0.000, B 0.000, C 0.000 }
gfCNCPoint4[16067] = {X 492.3835, Y 7.9502, Z -5.5000, A 0.000, B 0.000, C 0.000 }
gfCNCPoint4[16068] = {X 502.2063, Y 7.9502, Z -5.5000, A 0.000, B 0.000, C 0.000 }
gfCNCPoint4[16069] = {X 502.7389, Y 7.9544, Z -5.5000, A 0.000, B 0.000, C 0.000 }
gfCNCPoint4[16070] = {X 503.6730, Y 8.0665, Z -5.5000, A 0.000, B 0.000, C 0.000 }
gfCNCPoint4[16071] = {X 504.5592, Y 8.3827, Z -5.5000, A 0.000, B 0.000, C 0.000 }
gfCNCPoint4[16072] = {X 505.3533, Y 8.8873, Z -5.5000, A 0.000, B 0.000, C 0.000 }
gfCNCPoint4[16073] = {X 506.0160, Y 9.5552, Z -5.5000, A 0.000, B 0.000, C 0.000 }
gfCNCPoint4[16074] = {X 506.5144, Y 10.3532, Z -5.5000, A 0.000, B 0.000, C 0.000 }
gfCNCPoint4[16075] = {X 506.8237, Y 11.2419, Z -5.5000, A 0.000, B 0.000, C 0.000 }
gfCNCPoint4[16076] = {X 506.9285, Y 12.1769, Z -5.5000, A 0.000, B 0.000, C 0.000 }
gfCNCPoint4[16077] = {X 506.9285, Y 12.9782, Z -5.5000, A 0.000, B 0.000, C 0.000 }
gfCNCPoint4[16078] = {X 506.8271, Y 13.8998, Z -5.5000, A 0.000, B 0.000, C 0.000 }
gfCNCPoint4[16079] = {X 506.5278, Y 14.7773, Z -5.5000, A 0.000, B 0.000, C 0.000 }
gfCNCPoint4[16080] = {X 506.0449, Y 15.5688, Z -5.5000, A 0.000, B 0.000, C 0.000 }
gfCNCPoint4[16081] = {X 505.4015, Y 16.2364, Z -5.5000, A 0.000, B 0.000, C 0.000 }
gfCNCPoint4[16082] = {X 505.4014, Y 40.9508, Z -5.5000, A 0.000, B 0.000, C 0.000 }
gfCNCPoint4[16083] = {X 505.4297, Y 40.9741, Z -5.5000, A 0.000, B 0.000, C 0.000 }
gfCNCPoint4[16084] = {X 506.0561, Y 41.6327, Z -5.5000, A 0.000, B 0.000, C 0.000 }
gfCNCPoint4[16085] = {X 506.5278, Y 42.4096, Z -5.5000, A 0.000, B 0.000, C 0.000 }
gfCNCPoint4[16086] = {X 506.8231, Y 43.2692, Z -5.5000, A 0.000, B 0.000, C 0.000 }
gfCNCPoint4[16087] = {X 506.9283, Y 44.1720, Z -5.5000, A 0.000, B 0.000, C 0.000 }
gfCNCPoint4[16088] = {X 506.9285, Y 45.0000, Z -5.5000, A 0.000, B 0.000, C 0.000 }
gfCNCPoint4[16089] = {X 506.8222, Y 45.9435, Z -5.5000, A 0.000, B 0.000, C 0.000 }
gfCNCPoint4[16090] = {X 506.5086, Y 46.8397, Z -5.5000, A 0.000, B 0.000, C 0.000 }
gfCNCPoint4[16091] = {X 506.0035, Y 47.6436, Z -5.5000, A 0.000, B 0.000, C 0.000 }
gfCNCPoint4[16092] = {X 505.3321, Y 48.3150, Z -5.5000, A 0.000, B 0.000, C 0.000 }
gfCNCPoint4[16093] = {X 504.5282, Y 48.8201, Z -5.5000, A 0.000, B 0.000, C 0.000 }
gfCNCPoint4[16094] = {X 503.6320, Y 49.1337, Z -5.5000, A 0.000, B 0.000, C 0.000 }
gfCNCPoint4[16095] = {X 502.6885, Y 49.2400, Z -5.5000, A 0.000, B 0.000, C 0.000 }
gfCNCPoint4[16096] = {X 496.2450, Y 49.2400, Z -5.5000, A 0.000, B 0.000, C 0.000 }
gfCNCPoint4[16097] = {X 495.3062, Y 49.1348, Z -5.5000, A 0.000, B 0.000, C 0.000 }
gfCNCPoint4[16098] = {X 494.4140, Y 48.8242, Z -5.5000, A 0.000, B 0.000, C 0.000 }
gfCNCPoint4[16099] = {X 493.6127, Y 48.3239, Z -5.5000, A 0.000, B 0.000, C 0.000 }
gfCNCPoint4[16100] = {X 492.9420, Y 47.6585, Z -5.5000, A 0.000, B 0.000, C 0.000 }
gfCNCPoint4[16101] = {X 492.4354, Y 46.8612, Z -5.5000, A 0.000, B 0.000, C 0.000 }
gfCNCPoint4[16102] = {X 492.1178, Y 45.9714, Z -5.5000, A 0.000, B 0.000, C 0.000 }
gfCNCPoint4[16103] = {X 492.0052, Y 45.0335, Z -5.5000, A 0.000, B 0.000, C 0.000 }
gfCNCPoint4[16104] = {X 492.0054, Y 44.1505, Z -5.5000, A 0.000, B 0.000, C 0.000 }
gfCNCPoint4[16105] = {X 492.1159, Y 43.2454, Z -5.5000, A 0.000, B 0.000, C 0.000 }
gfCNCPoint4[16106] = {X 492.4173, Y 42.3850, Z -5.5000, A 0.000, B 0.000, C 0.000 }
gfCNCPoint4[16107] = {X 492.8957, Y 41.6088, Z -5.5000, A 0.000, B 0.000, C 0.000 }
gfCNCPoint4[16108] = {X 493.5290, Y 40.9529, Z -5.5000, A 0.000, B 0.000, C 0.000 }
gfCNCPoint4[16109] = {X 493.5290, Y 34.3938, Z -5.5000, A 0.000, B 0.000, C 0.000 }
gfCNCPoint4[16110] = {X 490.6759, Y 34.3938, Z -5.5000, A 0.000, B 0.000, C 0.000 }
gfCNCPoint4[16111] = {X 486.3531, Y 42.8122, Z -5.5000, A 0.000, B 0.000, C 0.000 }
gfCNCPoint4[16112] = {X 486.3697, Y 42.8569, Z -5.5000, A 0.000, B 0.000, C 0.000 }
gfCNCPoint4[16113] = {X 486.5322, Y 43.5050, Z -5.5000, A 0.000, B 0.000, C 0.000 }
gfCNCPoint4[16114] = {X 486.5908, Y 44.1706, Z -5.5000, A 0.000, B 0.000, C 0.000 }
gfCNCPoint4[16115] = {X 486.5910, Y 45.0000, Z -5.5000, A 0.000, B 0.000, C 0.000 }
gfCNCPoint4[16116] = {X 486.4847, Y 45.9435, Z -5.5000, A 0.000, B 0.000, C 0.000 }
gfCNCPoint4[16117] = {X 486.1711, Y 46.8397, Z -5.5000, A 0.000, B 0.000, C 0.000 }
gfCNCPoint4[16118] = {X 485.6660, Y 47.6436, Z -5.5000, A 0.000, B 0.000, C 0.000 }
gfCNCPoint4[16119] = {X 484.9946, Y 48.3150, Z -5.5000, A 0.000, B 0.000, C 0.000 }
gfCNCPoint4[16120] = {X 484.1907, Y 48.8201, Z -5.5000, A 0.000, B 0.000, C 0.000 }
gfCNCPoint4[16121] = {X 483.2945, Y 49.1337, Z -5.5000, A 0.000, B 0.000, C 0.000 }
gfCNCPoint4[16122] = {X 482.3510, Y 49.2400, Z -5.5000, A 0.000, B 0.000, C 0.000 }
gfCNCPoint4[16123] = {X 475.7650, Y 49.2400, Z -5.5000, A 0.000, B 0.000, C 0.000 }
gfCNCPoint4[16124] = {X 474.8215, Y 49.1337, Z -5.5000, A 0.000, B 0.000, C 0.000 }
gfCNCPoint4[16125] = {X 473.9253, Y 48.8201, Z -5.5000, A 0.000, B 0.000, C 0.000 }
gfCNCPoint4[16126] = {X 473.1214, Y 48.3150, Z -5.5000, A 0.000, B 0.000, C 0.000 }
gfCNCPoint4[16127] = {X 472.4500, Y 47.6436, Z -5.5000, A 0.000, B 0.000, C 0.000 }
gfCNCPoint4[16128] = {X 471.9449, Y 46.8397, Z -5.5000, A 0.000, B 0.000, C 0.000 }
gfCNCPoint4[16129] = {X 471.6313, Y 45.9436, Z -5.5000, A 0.000, B 0.000, C 0.000 }
gfCNCPoint4[16130] = {X 471.5250, Y 45.0001, Z -5.5000, A 0.000, B 0.000, C 0.000 }
gfCNCPoint4[16131] = {X 471.5254, Y 44.1505, Z -5.5000, A 0.000, B 0.000, C 0.000 }
gfCNCPoint4[16132] = {X 471.6223, Y 43.3054, Z -5.5000, A 0.000, B 0.000, C 0.000 }
gfCNCPoint4[16133] = {X 471.8860, Y 42.4967, Z -5.5000, A 0.000, B 0.000, C 0.000 }
gfCNCPoint4[16134] = {X 472.3057, Y 41.7570, Z -5.5000, A 0.000, B 0.000, C 0.000 }
gfCNCPoint4[16135] = {X 472.8647, Y 41.1158, Z -5.5000, A 0.000, B 0.000, C 0.000 }
gfCNCPoint4[16136] = {X 473.5404, Y 40.5992, Z -5.5000, A 0.000, B 0.000, C 0.000 }
gfCNCPoint4[16137] = {X 474.3057, Y 40.2278, Z -5.5000, A 0.000, B 0.000, C 0.000 }
gfCNCPoint4[16138] = {X 478.3385, Y 32.3339, Z -5.5000, A 0.000, B 0.000, C 0.000 }
gfCNCPoint4[16139] = {X 477.0678, Y 31.4734, Z -5.5000, A 0.000, B 0.000, C 0.000 }
gfCNCPoint4[16140] = {X 475.9244, Y 30.4497, Z -5.5000, A 0.000, B 0.000, C 0.000 }
gfCNCPoint4[16141] = {X 474.9293, Y 29.2814, Z -5.5000, A 0.000, B 0.000, C 0.000 }
gfCNCPoint4[16142] = {X 474.1005, Y 27.9897, Z -5.5000, A 0.000, B 0.000, C 0.000 }
gfCNCPoint4[16143] = {X 473.4531, Y 26.5983, Z -5.5000, A 0.000, B 0.000, C 0.000 }
gfCNCPoint4[16144] = {X 472.9989, Y 25.1323, Z -5.5000, A 0.000, B 0.000, C 0.000 }
gfCNCPoint4[16145] = {X 472.6863, Y 23.4573, Z -5.5000, A 0.000, B 0.000, C 0.000 }
gfCNCPoint4[16146] = {X 472.5465, Y 21.7591, Z -5.5000, A 0.000, B 0.000, C 0.000 }
gfCNCPoint4[16147] = {X 472.5811, Y 20.0555, Z -5.5000, A 0.000, B 0.000, C 0.000 }
gfCNCPoint4[16148] = {X 472.7896, Y 18.3643, Z -5.5000, A 0.000, B 0.000, C 0.000 }
gfCNCPoint4[16149] = {X 473.1698, Y 16.7033, Z -5.5000, A 0.000, B 0.000, C 0.000 }
gfCNCPoint4[16150] = {X 473.7089, Y 15.1987, Z -5.5000, A 0.000, B 0.000, C 0.000 }
gfCNCPoint4[16151] = {X 474.4473, Y 13.7811, Z -5.5000, A 0.000, B 0.000, C 0.000 }
gfCNCPoint4[16152] = {X 475.3711, Y 12.4768, Z -5.5000, A 0.000, B 0.000, C 0.000 }
gfCNCPoint4[16153] = {X 476.4634, Y 11.3100, Z -5.5000, A 0.000, B 0.000, C 0.000 }
gfCNCPoint4[16154] = {X 477.7039, Y 10.3021, Z -5.5000, A 0.000, B 0.000, C 0.000 }
gfCNCPoint4[16155] = {X 479.0697, Y 9.4719, Z -5.5000, A 0.000, B 0.000, C 0.000 }
gfCNCPoint4[16156] = {X 480.5355, Y 8.8346, Z -5.5000, A 0.000, B 0.000, C 0.000 }
gfCNCPoint4[16157] = {X 482.0742, Y 8.4022, Z -5.5000, A 0.000, B 0.000, C 0.000 }
gfCNCPoint4[16158] = {X 484.1638, Y 8.0766, Z -5.5000, A 0.000, B 0.000, C 0.000 }
gfCNCPoint4[16159] = {X 486.2756, Y 7.9624, Z -5.5000, A 0.000, B 0.000, C 0.000 }
gfCNCPoint4[16160] = {X 486.9686, Y 7.9502, Z -5.5000, A 0.000, B 0.000, C 0.000 }
gfCNCPoint4[16161] = {X 492.3835, Y 7.9502, Z -5.5000, A 0.000, B 0.000, C 0.000 }
gfCNCPoint4[16162] = {X 492.3835, Y 3.9502, Z -5.5000, A 0.000, B 0.000, C 0.000 }
gfCNCPoint4[16163] = {X 492.3835, Y 8.0302, Z -5.5000, A 0.000, B 0.000, C 0.000 }
gfCNCPoint4[16164] = {X 502.2059, Y 8.0302, Z -5.5000, A 0.000, B 0.000, C 0.000 }
gfCNCPoint4[16165] = {X 502.7382, Y 8.0344, Z -5.5000, A 0.000, B 0.000, C 0.000 }
gfCNCPoint4[16166] = {X 503.6547, Y 8.1444, Z -5.5000, A 0.000, B 0.000, C 0.000 }
gfCNCPoint4[16167] = {X 504.5241, Y 8.4546, Z -5.5000, A 0.000, B 0.000, C 0.000 }
gfCNCPoint4[16168] = {X 505.3032, Y 8.9496, Z -5.5000, A 0.000, B 0.000, C 0.000 }
gfCNCPoint4[16169] = {X 505.9533, Y 9.6049, Z -5.5000, A 0.000, B 0.000, C 0.000 }
gfCNCPoint4[16170] = {X 506.4422, Y 10.3878, Z -5.5000, A 0.000, B 0.000, C 0.000 }
gfCNCPoint4[16171] = {X 506.7457, Y 11.2596, Z -5.5000, A 0.000, B 0.000, C 0.000 }
gfCNCPoint4[16172] = {X 506.8485, Y 12.1769, Z -5.5000, A 0.000, B 0.000, C 0.000 }
gfCNCPoint4[16173] = {X 506.8485, Y 12.9782, Z -5.5000, A 0.000, B 0.000, C 0.000 }
gfCNCPoint4[16174] = {X 506.7470, Y 13.8915, Z -5.5000, A 0.000, B 0.000, C 0.000 }
gfCNCPoint4[16175] = {X 506.4474, Y 14.7603, Z -5.5000, A 0.000, B 0.000, C 0.000 }
gfCNCPoint4[16176] = {X 505.9644, Y 15.5420, Z -5.5000, A 0.000, B 0.000, C 0.000 }
gfCNCPoint4[16177] = {X 505.3215, Y 16.1987, Z -5.5000, A 0.000, B 0.000, C 0.000 }
gfCNCPoint4[16178] = {X 505.3214, Y 40.9890, Z -5.5000, A 0.000, B 0.000, C 0.000 }
gfCNCPoint4[16179] = {X 505.3680, Y 41.0267, Z -5.5000, A 0.000, B 0.000, C 0.000 }
gfCNCPoint4[16180] = {X 505.9866, Y 41.6735, Z -5.5000, A 0.000, B 0.000, C 0.000 }
gfCNCPoint4[16181] = {X 506.4526, Y 42.4376, Z -5.5000, A 0.000, B 0.000, C 0.000 }
gfCNCPoint4[16182] = {X 506.7443, Y 43.2838, Z -5.5000, A 0.000, B 0.000, C 0.000 }
gfCNCPoint4[16183] = {X 506.8483, Y 44.1727, Z -5.5000, A 0.000, B 0.000, C 0.000 }
gfCNCPoint4[16184] = {X 506.8485, Y 45.0000, Z -5.5000, A 0.000, B 0.000, C 0.000 }
gfCNCPoint4[16185] = {X 506.7442, Y 45.9257, Z -5.5000, A 0.000, B 0.000, C 0.000 }
gfCNCPoint4[16186] = {X 506.4365, Y 46.8050, Z -5.5000, A 0.000, B 0.000, C 0.000 }
gfCNCPoint4[16187] = {X 505.9409, Y 47.5937, Z -5.5000, A 0.000, B 0.000, C 0.000 }
gfCNCPoint4[16188] = {X 505.2822, Y 48.2524, Z -5.5000, A 0.000, B 0.000, C 0.000 }
gfCNCPoint4[16189] = {X 504.4934, Y 48.7480, Z -5.5000, A 0.000, B 0.000, C 0.000 }
gfCNCPoint4[16190] = {X 503.6142, Y 49.0557, Z -5.5000, A 0.000, B 0.000, C 0.000 }
gfCNCPoint4[16191] = {X 502.6885, Y 49.1600, Z -5.5000, A 0.000, B 0.000, C 0.000 }
gfCNCPoint4[16192] = {X 496.2450, Y 49.1600, Z -5.5000, A 0.000, B 0.000, C 0.000 }
gfCNCPoint4[16193] = {X 495.3239, Y 49.0567, Z -5.5000, A 0.000, B 0.000, C 0.000 }
gfCNCPoint4[16194] = {X 494.4485, Y 48.7521, Z -5.5000, A 0.000, B 0.000, C 0.000 }
gfCNCPoint4[16195] = {X 493.6623, Y 48.2612, Z -5.5000, A 0.000, B 0.000, C 0.000 }
gfCNCPoint4[16196] = {X 493.0043, Y 47.6084, Z -5.5000, A 0.000, B 0.000, C 0.000 }
gfCNCPoint4[16197] = {X 492.5072, Y 46.8261, Z -5.5000, A 0.000, B 0.000, C 0.000 }
gfCNCPoint4[16198] = {X 492.1957, Y 45.9531, Z -5.5000, A 0.000, B 0.000, C 0.000 }
gfCNCPoint4[16199] = {X 492.0852, Y 45.0328, Z -5.5000, A 0.000, B 0.000, C 0.000 }
gfCNCPoint4[16200] = {X 492.0854, Y 44.1516, Z -5.5000, A 0.000, B 0.000, C 0.000 }
gfCNCPoint4[16201] = {X 492.1960, Y 43.2545, Z -5.5000, A 0.000, B 0.000, C 0.000 }
gfCNCPoint4[16202] = {X 492.4976, Y 42.4026, Z -5.5000, A 0.000, B 0.000, C 0.000 }
gfCNCPoint4[16203] = {X 492.9762, Y 41.6358, Z -5.5000, A 0.000, B 0.000, C 0.000 }
gfCNCPoint4[16204] = {X 493.6090, Y 40.9906, Z -5.5000, A 0.000, B 0.000, C 0.000 }
gfCNCPoint4[16205] = {X 493.6090, Y 34.3138, Z -5.5000, A 0.000, B 0.000, C 0.000 }
gfCNCPoint4[16206] = {X 490.6271, Y 34.3138, Z -5.5000, A 0.000, B 0.000, C 0.000 }
gfCNCPoint4[16207] = {X 486.2658, Y 42.8071, Z -5.5000, A 0.000, B 0.000, C 0.000 }
gfCNCPoint4[16208] = {X 486.2943, Y 42.8836, Z -5.5000, A 0.000, B 0.000, C 0.000 }
gfCNCPoint4[16209] = {X 486.4534, Y 43.5189, Z -5.5000, A 0.000, B 0.000, C 0.000 }
gfCNCPoint4[16210] = {X 486.5108, Y 44.1713, Z -5.5000, A 0.000, B 0.000, C 0.000 }
gfCNCPoint4[16211] = {X 486.5110, Y 45.0000, Z -5.5000, A 0.000, B 0.000, C 0.000 }
gfCNCPoint4[16212] = {X 486.4067, Y 45.9257, Z -5.5000, A 0.000, B 0.000, C 0.000 }
gfCNCPoint4[16213] = {X 486.0990, Y 46.8050, Z -5.5000, A 0.000, B 0.000, C 0.000 }
gfCNCPoint4[16214] = {X 485.6034, Y 47.5937, Z -5.5000, A 0.000, B 0.000, C 0.000 }
gfCNCPoint4[16215] = {X 484.9447, Y 48.2524, Z -5.5000, A 0.000, B 0.000, C 0.000 }
gfCNCPoint4[16216] = {X 484.1560, Y 48.7480, Z -5.5000, A 0.000, B 0.000, C 0.000 }
gfCNCPoint4[16217] = {X 483.2767, Y 49.0557, Z -5.5000, A 0.000, B 0.000, C 0.000 }
gfCNCPoint4[16218] = {X 482.3510, Y 49.1600, Z -5.5000, A 0.000, B 0.000, C 0.000 }
gfCNCPoint4[16219] = {X 475.7650, Y 49.1600, Z -5.5000, A 0.000, B 0.000, C 0.000 }
gfCNCPoint4[16220] = {X 474.8393, Y 49.0557, Z -5.5000, A 0.000, B 0.000, C 0.000 }
gfCNCPoint4[16221] = {X 473.9600, Y 48.7480, Z -5.5000, A 0.000, B 0.000, C 0.000 }
gfCNCPoint4[16222] = {X 473.1713, Y 48.2524, Z -5.5000, A 0.000, B 0.000, C 0.000 }
gfCNCPoint4[16223] = {X 472.5126, Y 47.5937, Z -5.5000, A 0.000, B 0.000, C 0.000 }
gfCNCPoint4[16224] = {X 472.0169, Y 46.8050, Z -5.5000, A 0.000, B 0.000, C 0.000 }
gfCNCPoint4[16225] = {X 471.7093, Y 45.9257, Z -5.5000, A 0.000, B 0.000, C 0.000 }
gfCNCPoint4[16226] = {X 471.6050, Y 45.0000, Z -5.5000, A 0.000, B 0.000, C 0.000 }
gfCNCPoint4[16227] = {X 471.6054, Y 44.1516, Z -5.5000, A 0.000, B 0.000, C 0.000 }
gfCNCPoint4[16228] = {X 471.7016, Y 43.3174, Z -5.5000, A 0.000, B 0.000, C 0.000 }
gfCNCPoint4[16229] = {X 471.9634, Y 42.5195, Z -5.5000, A 0.000, B 0.000, C 0.000 }
gfCNCPoint4[16230] = {X 472.3801, Y 41.7905, Z -5.5000, A 0.000, B 0.000, C 0.000 }
gfCNCPoint4[16231] = {X 472.9347, Y 41.1600, Z -5.5000, A 0.000, B 0.000, C 0.000 }
gfCNCPoint4[16232] = {X 473.6046, Y 40.6537, Z -5.5000, A 0.000, B 0.000, C 0.000 }
gfCNCPoint4[16233] = {X 474.3626, Y 40.2923, Z -5.5000, A 0.000, B 0.000, C 0.000 }
gfCNCPoint4[16234] = {X 478.4443, Y 32.3027, Z -5.5000, A 0.000, B 0.000, C 0.000 }
gfCNCPoint4[16235] = {X 477.1668, Y 31.4490, Z -5.5000, A 0.000, B 0.000, C 0.000 }
gfCNCPoint4[16236] = {X 476.0170, Y 30.4298, Z -5.5000, A 0.000, B 0.000, C 0.000 }
gfCNCPoint4[16237] = {X 475.0161, Y 29.2640, Z -5.5000, A 0.000, B 0.000, C 0.000 }
gfCNCPoint4[16238] = {X 474.1827, Y 27.9732, Z -5.5000, A 0.000, B 0.000, C 0.000 }
gfCNCPoint4[16239] = {X 473.5322, Y 26.5812, Z -5.5000, A 0.000, B 0.000, C 0.000 }
gfCNCPoint4[16240] = {X 473.0767, Y 25.1137, Z -5.5000, A 0.000, B 0.000, C 0.000 }
gfCNCPoint4[16241] = {X 472.7656, Y 23.4467, Z -5.5000, A 0.000, B 0.000, C 0.000 }
gfCNCPoint4[16242] = {X 472.6265, Y 21.7567, Z -5.5000, A 0.000, B 0.000, C 0.000 }
gfCNCPoint4[16243] = {X 472.6609, Y 20.0612, Z -5.5000, A 0.000, B 0.000, C 0.000 }
gfCNCPoint4[16244] = {X 472.8684, Y 18.3782, Z -5.5000, A 0.000, B 0.000, C 0.000 }
gfCNCPoint4[16245] = {X 473.2468, Y 16.7251, Z -5.5000, A 0.000, B 0.000, C 0.000 }
gfCNCPoint4[16246] = {X 473.7822, Y 15.2307, Z -5.5000, A 0.000, B 0.000, C 0.000 }
gfCNCPoint4[16247] = {X 474.5155, Y 13.8228, Z -5.5000, A 0.000, B 0.000, C 0.000 }
gfCNCPoint4[16248] = {X 475.4331, Y 12.5274, Z -5.5000, A 0.000, B 0.000, C 0.000 }
gfCNCPoint4[16249] = {X 476.5179, Y 11.3685, Z -5.5000, A 0.000, B 0.000, C 0.000 }
gfCNCPoint4[16250] = {X 477.7500, Y 10.3675, Z -5.5000, A 0.000, B 0.000, C 0.000 }
gfCNCPoint4[16251] = {X 479.1065, Y 9.5429, Z -5.5000, A 0.000, B 0.000, C 0.000 }
gfCNCPoint4[16252] = {X 480.5623, Y 8.9100, Z -5.5000, A 0.000, B 0.000, C 0.000 }
gfCNCPoint4[16253] = {X 482.0906, Y 8.4805, Z -5.5000, A 0.000, B 0.000, C 0.000 }
gfCNCPoint4[16254] = {X 484.1725, Y 8.1562, Z -5.5000, A 0.000, B 0.000, C 0.000 }
gfCNCPoint4[16255] = {X 486.2765, Y 8.0424, Z -5.5000, A 0.000, B 0.000, C 0.000 }
gfCNCPoint4[16256] = {X 486.9693, Y 8.0302, Z -5.5000, A 0.000, B 0.000, C 0.000 }
gfCNCPoint4[16257] = {X 492.3835, Y 8.0302, Z -5.5000, A 0.000, B 0.000, C 0.000 }
gfCNCPoint4[16258] = {X 492.3835, Y 4.0302, Z -5.5000, A 0.000, B 0.000, C 0.000 }
gfCNCPoint4[16259] = {X 492.3835, Y 8.1102, Z -5.5000, A 0.000, B 0.000, C 0.000 }
gfCNCPoint4[16260] = {X 502.2056, Y 8.1102, Z -5.5000, A 0.000, B 0.000, C 0.000 }
gfCNCPoint4[16261] = {X 502.7376, Y 8.1144, Z -5.5000, A 0.000, B 0.000, C 0.000 }
gfCNCPoint4[16262] = {X 503.6364, Y 8.2223, Z -5.5000, A 0.000, B 0.000, C 0.000 }
gfCNCPoint4[16263] = {X 504.4890, Y 8.5265, Z -5.5000, A 0.000, B 0.000, C 0.000 }
gfCNCPoint4[16264] = {X 505.2530, Y 9.0119, Z -5.5000, A 0.000, B 0.000, C 0.000 }
gfCNCPoint4[16265] = {X 505.8906, Y 9.6545, Z -5.5000, A 0.000, B 0.000, C 0.000 }
gfCNCPoint4[16266] = {X 506.3701, Y 10.4223, Z -5.5000, A 0.000, B 0.000, C 0.000 }
gfCNCPoint4[16267] = {X 506.6676, Y 11.2773, Z -5.5000, A 0.000, B 0.000, C 0.000 }
gfCNCPoint4[16268] = {X 506.7685, Y 12.1769, Z -5.5000, A 0.000, B 0.000, C 0.000 }
gfCNCPoint4[16269] = {X 506.7685, Y 12.9782, Z -5.5000, A 0.000, B 0.000, C 0.000 }
gfCNCPoint4[16270] = {X 506.6668, Y 13.8831, Z -5.5000, A 0.000, B 0.000, C 0.000 }
gfCNCPoint4[16271] = {X 506.3670, Y 14.7430, Z -5.5000, A 0.000, B 0.000, C 0.000 }
gfCNCPoint4[16272] = {X 505.8838, Y 15.5150, Z -5.5000, A 0.000, B 0.000, C 0.000 }
gfCNCPoint4[16273] = {X 505.2415, Y 16.1606, Z -5.5000, A 0.000, B 0.000, C 0.000 }
gfCNCPoint4[16274] = {X 505.2414, Y 41.0272, Z -5.5000, A 0.000, B 0.000, C 0.000 }
gfCNCPoint4[16275] = {X 505.3177, Y 41.0889, Z -5.5000, A 0.000, B 0.000, C 0.000 }
gfCNCPoint4[16276] = {X 505.9239, Y 41.7232, Z -5.5000, A 0.000, B 0.000, C 0.000 }
gfCNCPoint4[16277] = {X 506.3805, Y 42.4724, Z -5.5000, A 0.000, B 0.000, C 0.000 }
gfCNCPoint4[16278] = {X 506.6664, Y 43.3019, Z -5.5000, A 0.000, B 0.000, C 0.000 }
gfCNCPoint4[16279] = {X 506.7683, Y 44.1734, Z -5.5000, A 0.000, B 0.000, C 0.000 }
gfCNCPoint4[16280] = {X 506.7685, Y 45.0000, Z -5.5000, A 0.000, B 0.000, C 0.000 }
gfCNCPoint4[16281] = {X 506.6662, Y 45.9079, Z -5.5000, A 0.000, B 0.000, C 0.000 }
gfCNCPoint4[16282] = {X 506.3644, Y 46.7702, Z -5.5000, A 0.000, B 0.000, C 0.000 }
gfCNCPoint4[16283] = {X 505.8784, Y 47.5438, Z -5.5000, A 0.000, B 0.000, C 0.000 }
gfCNCPoint4[16284] = {X 505.2323, Y 48.1899, Z -5.5000, A 0.000, B 0.000, C 0.000 }
gfCNCPoint4[16285] = {X 504.4587, Y 48.6760, Z -5.5000, A 0.000, B 0.000, C 0.000 }
gfCNCPoint4[16286] = {X 503.5964, Y 48.9777, Z -5.5000, A 0.000, B 0.000, C 0.000 }
gfCNCPoint4[16287] = {X 502.6885, Y 49.0800, Z -5.5000, A 0.000, B 0.000, C 0.000 }
gfCNCPoint4[16288] = {X 496.2450, Y 49.0800, Z -5.5000, A 0.000, B 0.000, C 0.000 }
gfCNCPoint4[16289] = {X 495.3416, Y 48.9787, Z -5.5000, A 0.000, B 0.000, C 0.000 }
gfCNCPoint4[16290] = {X 494.4831, Y 48.6799, Z -5.5000, A 0.000, B 0.000, C 0.000 }
gfCNCPoint4[16291] = {X 493.7120, Y 48.1985, Z -5.5000, A 0.000, B 0.000, C 0.000 }
gfCNCPoint4[16292] = {X 493.0667, Y 47.5582, Z -5.5000, A 0.000, B 0.000, C 0.000 }
gfCNCPoint4[16293] = {X 492.5791, Y 46.7909, Z -5.5000, A 0.000, B 0.000, C 0.000 }
gfCNCPoint4[16294] = {X 492.2736, Y 45.9348, Z -5.5000, A 0.000, B 0.000, C 0.000 }
gfCNCPoint4[16295] = {X 492.1652, Y 45.0322, Z -5.5000, A 0.000, B 0.000, C 0.000 }
gfCNCPoint4[16296] = {X 492.1654, Y 44.1527, Z -5.5000, A 0.000, B 0.000, C 0.000 }
gfCNCPoint4[16297] = {X 492.2760, Y 43.2637, Z -5.5000, A 0.000, B 0.000, C 0.000 }
gfCNCPoint4[16298] = {X 492.5779, Y 42.4203, Z -5.5000, A 0.000, B 0.000, C 0.000 }
gfCNCPoint4[16299] = {X 493.0566, Y 41.6631, Z -5.5000, A 0.000, B 0.000, C 0.000 }
gfCNCPoint4[16300] = {X 493.6890, Y 41.0287, Z -5.5000, A 0.000, B 0.000, C 0.000 }
gfCNCPoint4[16301] = {X 493.6890, Y 34.2338, Z -5.5000, A 0.000, B 0.000, C 0.000 }
gfCNCPoint4[16302] = {X 490.5782, Y 34.2338, Z -5.5000, A 0.000, B 0.000, C 0.000 }
gfCNCPoint4[16303] = {X 486.1785, Y 42.8019, Z -5.5000, A 0.000, B 0.000, C 0.000 }
gfCNCPoint4[16304] = {X 486.2189, Y 42.9103, Z -5.5000, A 0.000, B 0.000, C 0.000 }
gfCNCPoint4[16305] = {X 486.3746, Y 43.5328, Z -5.5000, A 0.000, B 0.000, C 0.000 }
gfCNCPoint4[16306] = {X 486.4309, Y 44.1720, Z -5.5000, A 0.000, B 0.000, C 0.000 }
gfCNCPoint4[16307] = {X 486.4310, Y 45.0000, Z -5.5000, A 0.000, B 0.000, C 0.000 }
gfCNCPoint4[16308] = {X 486.3287, Y 45.9079, Z -5.5000, A 0.000, B 0.000, C 0.000 }
gfCNCPoint4[16309] = {X 486.0270, Y 46.7702, Z -5.5000, A 0.000, B 0.000, C 0.000 }
gfCNCPoint4[16310] = {X 485.5409, Y 47.5438, Z -5.5000, A 0.000, B 0.000, C 0.000 }
gfCNCPoint4[16311] = {X 484.8949, Y 48.1899, Z -5.5000, A 0.000, B 0.000, C 0.000 }
gfCNCPoint4[16312] = {X 484.1213, Y 48.6760, Z -5.5000, A 0.000, B 0.000, C 0.000 }
gfCNCPoint4[16313] = {X 483.2589, Y 48.9777, Z -5.5000, A 0.000, B 0.000, C 0.000 }
gfCNCPoint4[16314] = {X 482.3510, Y 49.0800, Z -5.5000, A 0.000, B 0.000, C 0.000 }
gfCNCPoint4[16315] = {X 475.7650, Y 49.0800, Z -5.5000, A 0.000, B 0.000, C 0.000 }
gfCNCPoint4[16316] = {X 474.8571, Y 48.9777, Z -5.5000, A 0.000, B 0.000, C 0.000 }
gfCNCPoint4[16317] = {X 473.9947, Y 48.6760, Z -5.5000, A 0.000, B 0.000, C 0.000 }
gfCNCPoint4[16318] = {X 473.2211, Y 48.1899, Z -5.5000, A 0.000, B 0.000, C 0.000 }
gfCNCPoint4[16319] = {X 472.5751, Y 47.5438, Z -5.5000, A 0.000, B 0.000, C 0.000 }
gfCNCPoint4[16320] = {X 472.0890, Y 46.7702, Z -5.5000, A 0.000, B 0.000, C 0.000 }
gfCNCPoint4[16321] = {X 471.7873, Y 45.9079, Z -5.5000, A 0.000, B 0.000, C 0.000 }
gfCNCPoint4[16322] = {X 471.6850, Y 45.0000, Z -5.5000, A 0.000, B 0.000, C 0.000 }
gfCNCPoint4[16323] = {X 471.6853, Y 44.1527, Z -5.5000, A 0.000, B 0.000, C 0.000 }
gfCNCPoint4[16324] = {X 471.7809, Y 43.3294, Z -5.5000, A 0.000, B 0.000, C 0.000 }
gfCNCPoint4[16325] = {X 472.0408, Y 42.5424, Z -5.5000, A 0.000, B 0.000, C 0.000 }
gfCNCPoint4[16326] = {X 472.4544, Y 41.8242, Z -5.5000, A 0.000, B 0.000, C 0.000 }
gfCNCPoint4[16327] = {X 473.0046, Y 41.2044, Z -5.5000, A 0.000, B 0.000, C 0.000 }
gfCNCPoint4[16328] = {X 473.6687, Y 40.7085, Z -5.5000, A 0.000, B 0.000, C 0.000 }
gfCNCPoint4[16329] = {X 474.4193, Y 40.3571, Z -5.5000, A 0.000, B 0.000, C 0.000 }
gfCNCPoint4[16330] = {X 478.5503, Y 32.2710, Z -5.5000, A 0.000, B 0.000, C 0.000 }
gfCNCPoint4[16331] = {X 477.2660, Y 31.4243, Z -5.5000, A 0.000, B 0.000, C 0.000 }
gfCNCPoint4[16332] = {X 476.1096, Y 30.4098, Z -5.5000, A 0.000, B 0.000, C 0.000 }
gfCNCPoint4[16333] = {X 475.1030, Y 29.2466, Z -5.5000, A 0.000, B 0.000, C 0.000 }
gfCNCPoint4[16334] = {X 474.2650, Y 27.9566, Z -5.5000, A 0.000, B 0.000, C 0.000 }
gfCNCPoint4[16335] = {X 473.6114, Y 26.5640, Z -5.5000, A 0.000, B 0.000, C 0.000 }
gfCNCPoint4[16336] = {X 473.1545, Y 25.0951, Z -5.5000, A 0.000, B 0.000, C 0.000 }
gfCNCPoint4[16337] = {X 472.8449, Y 23.4361, Z -5.5000, A 0.000, B 0.000, C 0.000 }
gfCNCPoint4[16338] = {X 472.7065, Y 21.7542, Z -5.5000, A 0.000, B 0.000, C 0.000 }
gfCNCPoint4[16339] = {X 472.7407, Y 20.0669, Z -5.5000, A 0.000, B 0.000, C 0.000 }
gfCNCPoint4[16340] = {X 472.9471, Y 18.3920, Z -5.5000, A 0.000, B 0.000, C 0.000 }
gfCNCPoint4[16341] = {X 473.3237, Y 16.7469, Z -5.5000, A 0.000, B 0.000, C 0.000 }
gfCNCPoint4[16342] = {X 473.8555, Y 15.2628, Z -5.5000, A 0.000, B 0.000, C 0.000 }
gfCNCPoint4[16343] = {X 474.5838, Y 13.8645, Z -5.5000, A 0.000, B 0.000, C 0.000 }
gfCNCPoint4[16344] = {X 475.4951, Y 12.5780, Z -5.5000, A 0.000, B 0.000, C 0.000 }
gfCNCPoint4[16345] = {X 476.5725, Y 11.4270, Z -5.5000, A 0.000, B 0.000, C 0.000 }
gfCNCPoint4[16346] = {X 477.7961, Y 10.4328, Z -5.5000, A 0.000, B 0.000, C 0.000 }
gfCNCPoint4[16347] = {X 479.1433, Y 9.6139, Z -5.5000, A 0.000, B 0.000, C 0.000 }
gfCNCPoint4[16348] = {X 480.5892, Y 8.9854, Z -5.5000, A 0.000, B 0.000, C 0.000 }
gfCNCPoint4[16349] = {X 482.1069, Y 8.5588, Z -5.5000, A 0.000, B 0.000, C 0.000 }
gfCNCPoint4[16350] = {X 484.1811, Y 8.2357, Z -5.5000, A 0.000, B 0.000, C 0.000 }
gfCNCPoint4[16351] = {X 486.2773, Y 8.1224, Z -5.5000, A 0.000, B 0.000, C 0.000 }
gfCNCPoint4[16352] = {X 486.9700, Y 8.1102, Z -5.5000, A 0.000, B 0.000, C 0.000 }
gfCNCPoint4[16353] = {X 492.3835, Y 8.1102, Z -5.5000, A 0.000, B 0.000, C 0.000 }
gfCNCPoint4[16354] = {X 492.3835, Y 4.1102, Z -5.5000, A 0.000, B 0.000, C 0.000 }
gfCNCPoint4[16355] = {X 492.3835, Y 8.1902, Z -5.5000, A 0.000, B 0.000, C 0.000 }
gfCNCPoint4[16356] = {X 502.2053, Y 8.1902, Z -5.5000, A 0.000, B 0.000, C 0.000 }
gfCNCPoint4[16357] = {X 502.7370, Y 8.1944, Z -5.5000, A 0.000, B 0.000, C 0.000 }
gfCNCPoint4[16358] = {X 503.6181, Y 8.3001, Z -5.5000, A 0.000, B 0.000, C 0.000 }
gfCNCPoint4[16359] = {X 504.4539, Y 8.5984, Z -5.5000, A 0.000, B 0.000, C 0.000 }
gfCNCPoint4[16360] = {X 505.2029, Y 9.0743, Z -5.5000, A 0.000, B 0.000, C 0.000 }
gfCNCPoint4[16361] = {X 505.8279, Y 9.7042, Z -5.5000, A 0.000, B 0.000, C 0.000 }
gfCNCPoint4[16362] = {X 506.2979, Y 10.4569, Z -5.5000, A 0.000, B 0.000, C 0.000 }
gfCNCPoint4[16363] = {X 506.5896, Y 11.2950, Z -5.5000, A 0.000, B 0.000, C 0.000 }
gfCNCPoint4[16364] = {X 506.6885, Y 12.1769, Z -5.5000, A 0.000, B 0.000, C 0.000 }
gfCNCPoint4[16365] = {X 506.6883, Y 13.0192, Z -5.5000, A 0.000, B 0.000, C 0.000 }
gfCNCPoint4[16366] = {X 506.5797, Y 13.9047, Z -5.5000, A 0.000, B 0.000, C 0.000 }
gfCNCPoint4[16367] = {X 506.2775, Y 14.7441, Z -5.5000, A 0.000, B 0.000, C 0.000 }
gfCNCPoint4[16368] = {X 505.7968, Y 15.4956, Z -5.5000, A 0.000, B 0.000, C 0.000 }
gfCNCPoint4[16369] = {X 505.1615, Y 16.1219, Z -5.5000, A 0.000, B 0.000, C 0.000 }
gfCNCPoint4[16370] = {X 505.1614, Y 41.0653, Z -5.5000, A 0.000, B 0.000, C 0.000 }
gfCNCPoint4[16371] = {X 505.3003, Y 41.1792, Z -5.5000, A 0.000, B 0.000, C 0.000 }
gfCNCPoint4[16372] = {X 505.8861, Y 41.8056, Z -5.5000, A 0.000, B 0.000, C 0.000 }
gfCNCPoint4[16373] = {X 506.3249, Y 42.5426, Z -5.5000, A 0.000, B 0.000, C 0.000 }
gfCNCPoint4[16374] = {X 506.5966, Y 43.3561, Z -5.5000, A 0.000, B 0.000, C 0.000 }
gfCNCPoint4[16375] = {X 506.6885, Y 44.2089, Z -5.5000, A 0.000, B 0.000, C 0.000 }
gfCNCPoint4[16376] = {X 506.6885, Y 45.0000, Z -5.5000, A 0.000, B 0.000, C 0.000 }
gfCNCPoint4[16377] = {X 506.5882, Y 45.8901, Z -5.5000, A 0.000, B 0.000, C 0.000 }
gfCNCPoint4[16378] = {X 506.2924, Y 46.7355, Z -5.5000, A 0.000, B 0.000, C 0.000 }
gfCNCPoint4[16379] = {X 505.8158, Y 47.4940, Z -5.5000, A 0.000, B 0.000, C 0.000 }
gfCNCPoint4[16380] = {X 505.1825, Y 48.1273, Z -5.5000, A 0.000, B 0.000, C 0.000 }
gfCNCPoint4[16381] = {X 504.4240, Y 48.6039, Z -5.5000, A 0.000, B 0.000, C 0.000 }
gfCNCPoint4[16382] = {X 503.5786, Y 48.8997, Z -5.5000, A 0.000, B 0.000, C 0.000 }
gfCNCPoint4[16383] = {X 502.6885, Y 49.0000, Z -5.5000, A 0.000, B 0.000, C 0.000 }
gfCNCPoint4[16384] = {X 496.2450, Y 49.0000, Z -5.5000, A 0.000, B 0.000, C 0.000 }
gfCNCPoint4[16385] = {X 495.3549, Y 48.8997, Z -5.5000, A 0.000, B 0.000, C 0.000 }
gfCNCPoint4[16386] = {X 494.5095, Y 48.6039, Z -5.5000, A 0.000, B 0.000, C 0.000 }
gfCNCPoint4[16387] = {X 493.7511, Y 48.1273, Z -5.5000, A 0.000, B 0.000, C 0.000 }
gfCNCPoint4[16388] = {X 493.1177, Y 47.4939, Z -5.5000, A 0.000, B 0.000, C 0.000 }
gfCNCPoint4[16389] = {X 492.6411, Y 46.7355, Z -5.5000, A 0.000, B 0.000, C 0.000 }
gfCNCPoint4[16390] = {X 492.3453, Y 45.8901, Z -5.5000, A 0.000, B 0.000, C 0.000 }
gfCNCPoint4[16391] = {X 492.2450, Y 45.0000, Z -5.5000, A 0.000, B 0.000, C 0.000 }
gfCNCPoint4[16392] = {X 492.2454, Y 44.1538, Z -5.5000, A 0.000, B 0.000, C 0.000 }
gfCNCPoint4[16393] = {X 492.3560, Y 43.2730, Z -5.5000, A 0.000, B 0.000, C 0.000 }
gfCNCPoint4[16394] = {X 492.6582, Y 42.4382, Z -5.5000, A 0.000, B 0.000, C 0.000 }
gfCNCPoint4[16395] = {X 493.1371, Y 41.6907, Z -5.5000, A 0.000, B 0.000, C 0.000 }
gfCNCPoint4[16396] = {X 493.7690, Y 41.0672, Z -5.5000, A 0.000, B 0.000, C 0.000 }
gfCNCPoint4[16397] = {X 493.7690, Y 34.1538, Z -5.5000, A 0.000, B 0.000, C 0.000 }
gfCNCPoint4[16398] = {X 490.7737, Y 34.1538, Z -5.5000, A 0.000, B 0.000, C 0.000 }
gfCNCPoint4[16399] = {X 490.5304, Y 34.1519, Z -5.5000, A 0.000, B 0.000, C 0.000 }
gfCNCPoint4[16400] = {X 486.2782, Y 42.4361, Z -5.5000, A 0.000, B 0.000, C 0.000 }
gfCNCPoint4[16401] = {X 486.0911, Y 42.7966, Z -5.5000, A 0.000, B 0.000, C 0.000 }
gfCNCPoint4[16402] = {X 486.1478, Y 42.9500, Z -5.5000, A 0.000, B 0.000, C 0.000 }
gfCNCPoint4[16403] = {X 486.2999, Y 43.5713, Z -5.5000, A 0.000, B 0.000, C 0.000 }
gfCNCPoint4[16404] = {X 486.3510, Y 44.2089, Z -5.5000, A 0.000, B 0.000, C 0.000 }
gfCNCPoint4[16405] = {X 486.3510, Y 45.0000, Z -5.5000, A 0.000, B 0.000, C 0.000 }
gfCNCPoint4[16406] = {X 486.2507, Y 45.8901, Z -5.5000, A 0.000, B 0.000, C 0.000 }
gfCNCPoint4[16407] = {X 485.9549, Y 46.7355, Z -5.5000, A 0.000, B 0.000, C 0.000 }
gfCNCPoint4[16408] = {X 485.4783, Y 47.4940, Z -5.5000, A 0.000, B 0.000, C 0.000 }
gfCNCPoint4[16409] = {X 484.8450, Y 48.1273, Z -5.5000, A 0.000, B 0.000, C 0.000 }
gfCNCPoint4[16410] = {X 484.0866, Y 48.6039, Z -5.5000, A 0.000, B 0.000, C 0.000 }
gfCNCPoint4[16411] = {X 483.2411, Y 48.8997, Z -5.5000, A 0.000, B 0.000, C 0.000 }
gfCNCPoint4[16412] = {X 482.3510, Y 49.0000, Z -5.5000, A 0.000, B 0.000, C 0.000 }
gfCNCPoint4[16413] = {X 475.7650, Y 49.0000, Z -5.5000, A 0.000, B 0.000, C 0.000 }
gfCNCPoint4[16414] = {X 474.8749, Y 48.8997, Z -5.5000, A 0.000, B 0.000, C 0.000 }
gfCNCPoint4[16415] = {X 474.0294, Y 48.6039, Z -5.5000, A 0.000, B 0.000, C 0.000 }
gfCNCPoint4[16416] = {X 473.2710, Y 48.1273, Z -5.5000, A 0.000, B 0.000, C 0.000 }
gfCNCPoint4[16417] = {X 472.6376, Y 47.4940, Z -5.5000, A 0.000, B 0.000, C 0.000 }
gfCNCPoint4[16418] = {X 472.1611, Y 46.7355, Z -5.5000, A 0.000, B 0.000, C 0.000 }
gfCNCPoint4[16419] = {X 471.8652, Y 45.8901, Z -5.5000, A 0.000, B 0.000, C 0.000 }
gfCNCPoint4[16420] = {X 471.7650, Y 45.0000, Z -5.5000, A 0.000, B 0.000, C 0.000 }
gfCNCPoint4[16421] = {X 471.7653, Y 44.1538, Z -5.5000, A 0.000, B 0.000, C 0.000 }
gfCNCPoint4[16422] = {X 471.8601, Y 43.3414, Z -5.5000, A 0.000, B 0.000, C 0.000 }
gfCNCPoint4[16423] = {X 472.1182, Y 42.5654, Z -5.5000, A 0.000, B 0.000, C 0.000 }
gfCNCPoint4[16424] = {X 472.5286, Y 41.8580, Z -5.5000, A 0.000, B 0.000, C 0.000 }
gfCNCPoint4[16425] = {X 473.0744, Y 41.2489, Z -5.5000, A 0.000, B 0.000, C 0.000 }
gfCNCPoint4[16426] = {X 473.7327, Y 40.7635, Z -5.5000, A 0.000, B 0.000, C 0.000 }
gfCNCPoint4[16427] = {X 474.4759, Y 40.4222, Z -5.5000, A 0.000, B 0.000, C 0.000 }
gfCNCPoint4[16428] = {X 478.6566, Y 32.2388, Z -5.5000, A 0.000, B 0.000, C 0.000 }
gfCNCPoint4[16429] = {X 477.3655, Y 31.3993, Z -5.5000, A 0.000, B 0.000, C 0.000 }
gfCNCPoint4[16430] = {X 476.2025, Y 30.3896, Z -5.5000, A 0.000, B 0.000, C 0.000 }
gfCNCPoint4[16431] = {X 475.1900, Y 29.2291, Z -5.5000, A 0.000, B 0.000, C 0.000 }
gfCNCPoint4[16432] = {X 474.3473, Y 27.9400, Z -5.5000, A 0.000, B 0.000, C 0.000 }
gfCNCPoint4[16433] = {X 473.6906, Y 26.5469, Z -5.5000, A 0.000, B 0.000, C 0.000 }
gfCNCPoint4[16434] = {X 473.2323, Y 25.0766, Z -5.5000, A 0.000, B 0.000, C 0.000 }
gfCNCPoint4[16435] = {X 472.9242, Y 23.4256, Z -5.5000, A 0.000, B 0.000, C 0.000 }
gfCNCPoint4[16436] = {X 472.7864, Y 21.7518, Z -5.5000, A 0.000, B 0.000, C 0.000 }
gfCNCPoint4[16437] = {X 472.8205, Y 20.0727, Z -5.5000, A 0.000, B 0.000, C 0.000 }
gfCNCPoint4[16438] = {X 473.0259, Y 18.4059, Z -5.5000, A 0.000, B 0.000, C 0.000 }
gfCNCPoint4[16439] = {X 473.4007, Y 16.7687, Z -5.5000, A 0.000, B 0.000, C 0.000 }
gfCNCPoint4[16440] = {X 473.9288, Y 15.2948, Z -5.5000, A 0.000, B 0.000, C 0.000 }
gfCNCPoint4[16441] = {X 474.6521, Y 13.9062, Z -5.5000, A 0.000, B 0.000, C 0.000 }
gfCNCPoint4[16442] = {X 475.5571, Y 12.6285, Z -5.5000, A 0.000, B 0.000, C 0.000 }
gfCNCPoint4[16443] = {X 476.6270, Y 11.4855, Z -5.5000, A 0.000, B 0.000, C 0.000 }
gfCNCPoint4[16444] = {X 477.8422, Y 10.4982, Z -5.5000, A 0.000, B 0.000, C 0.000 }
gfCNCPoint4[16445] = {X 479.1801, Y 9.6850, Z -5.5000, A 0.000, B 0.000, C 0.000 }
gfCNCPoint4[16446] = {X 480.6160, Y 9.0607, Z -5.5000, A 0.000, B 0.000, C 0.000 }
gfCNCPoint4[16447] = {X 482.1233, Y 8.6371, Z -5.5000, A 0.000, B 0.000, C 0.000 }
gfCNCPoint4[16448] = {X 484.1898, Y 8.3152, Z -5.5000, A 0.000, B 0.000, C 0.000 }
gfCNCPoint4[16449] = {X 486.2782, Y 8.2024, Z -5.5000, A 0.000, B 0.000, C 0.000 }
gfCNCPoint4[16450] = {X 486.9707, Y 8.1902, Z -5.5000, A 0.000, B 0.000, C 0.000 }
gfCNCPoint4[16451] = {X 492.3835, Y 8.1902, Z -5.5000, A 0.000, B 0.000, C 0.000 }
gfCNCPoint4[16452] = {X 492.3835, Y 4.1102, Z -5.5000, A 0.000, B 0.000, C 0.000 }
gfCNCPoint4[16453] = {X 492.3835, Y 4.1102, Z -2.5000, A 0.000, B 0.000, C 0.000 }
gfCNCPoint4[16454] = {X 492.3835, Y 4.1102, Z 11.0000, A 0.000, B 0.000, C 0.000 }
gfCNCPoint4[16455] = {X 533.9636, Y 3.7900, Z 11.0000, A 0.000, B 0.000, C 0.000 }
gfCNCPoint4[16456] = {X 533.9636, Y 3.7900, Z -2.5000, A 0.000, B 0.000, C 0.000 }
gfCNCPoint4[16457] = {X 533.9636, Y 3.7900, Z -5.5000, A 0.000, B 0.000, C 0.000 }
gfCNCPoint4[16458] = {X 533.9635, Y 7.8700, Z -5.5000, A 0.000, B 0.000, C 0.000 }
gfCNCPoint4[16459] = {X 543.7499, Y 7.8702, Z -5.5000, A 0.000, B 0.000, C 0.000 }
gfCNCPoint4[16460] = {X 544.7302, Y 7.9558, Z -5.5000, A 0.000, B 0.000, C 0.000 }
gfCNCPoint4[16461] = {X 545.6658, Y 8.2606, Z -5.5000, A 0.000, B 0.000, C 0.000 }
gfCNCPoint4[16462] = {X 546.5082, Y 8.7691, Z -5.5000, A 0.000, B 0.000, C 0.000 }
gfCNCPoint4[16463] = {X 547.2139, Y 9.4549, Z -5.5000, A 0.000, B 0.000, C 0.000 }
gfCNCPoint4[16464] = {X 547.7463, Y 10.2824, Z -5.5000, A 0.000, B 0.000, C 0.000 }
gfCNCPoint4[16465] = {X 548.0779, Y 11.2089, Z -5.5000, A 0.000, B 0.000, C 0.000 }
gfCNCPoint4[16466] = {X 548.1914, Y 12.1863, Z -5.5000, A 0.000, B 0.000, C 0.000 }
gfCNCPoint4[16467] = {X 548.1912, Y 13.0225, Z -5.5000, A 0.000, B 0.000, C 0.000 }
gfCNCPoint4[16468] = {X 548.0830, Y 13.9400, Z -5.5000, A 0.000, B 0.000, C 0.000 }
gfCNCPoint4[16469] = {X 547.7821, Y 14.8135, Z -5.5000, A 0.000, B 0.000, C 0.000 }
gfCNCPoint4[16470] = {X 547.3024, Y 15.6031, Z -5.5000, A 0.000, B 0.000, C 0.000 }
gfCNCPoint4[16471] = {X 546.6658, Y 16.2726, Z -5.5000, A 0.000, B 0.000, C 0.000 }
gfCNCPoint4[16472] = {X 546.6644, Y 40.9138, Z -5.5000, A 0.000, B 0.000, C 0.000 }
gfCNCPoint4[16473] = {X 546.6863, Y 40.9318, Z -5.5000, A 0.000, B 0.000, C 0.000 }
gfCNCPoint4[16474] = {X 547.3160, Y 41.6017, Z -5.5000, A 0.000, B 0.000, C 0.000 }
gfCNCPoint4[16475] = {X 547.7897, Y 42.3896, Z -5.5000, A 0.000, B 0.000, C 0.000 }
gfCNCPoint4[16476] = {X 548.0859, Y 43.2600, Z -5.5000, A 0.000, B 0.000, C 0.000 }
gfCNCPoint4[16477] = {X 548.1913, Y 44.1733, Z -5.5000, A 0.000, B 0.000, C 0.000 }
gfCNCPoint4[16478] = {X 548.1914, Y 45.0005, Z -5.5000, A 0.000, B 0.000, C 0.000 }
gfCNCPoint4[16479] = {X 548.0779, Y 45.9779, Z -5.5000, A 0.000, B 0.000, C 0.000 }
gfCNCPoint4[16480] = {X 547.7463, Y 46.9044, Z -5.5000, A 0.000, B 0.000, C 0.000 }
gfCNCPoint4[16481] = {X 547.2139, Y 47.7319, Z -5.5000, A 0.000, B 0.000, C 0.000 }
gfCNCPoint4[16482] = {X 546.5082, Y 48.4176, Z -5.5000, A 0.000, B 0.000, C 0.000 }
gfCNCPoint4[16483] = {X 545.6658, Y 48.9260, Z -5.5000, A 0.000, B 0.000, C 0.000 }
gfCNCPoint4[16484] = {X 544.7302, Y 49.2308, Z -5.5000, A 0.000, B 0.000, C 0.000 }
gfCNCPoint4[16485] = {X 543.7499, Y 49.3163, Z -5.5000, A 0.000, B 0.000, C 0.000 }
gfCNCPoint4[16486] = {X 524.0453, Y 49.3167, Z -5.5000, A 0.000, B 0.000, C 0.000 }
gfCNCPoint4[16487] = {X 523.4987, Y 49.9506, Z -5.5000, A 0.000, B 0.000, C 0.000 }
gfCNCPoint4[16488] = {X 522.8436, Y 50.4716, Z -5.5000, A 0.000, B 0.000, C 0.000 }
gfCNCPoint4[16489] = {X 522.1030, Y 50.8617, Z -5.5000, A 0.000, B 0.000, C 0.000 }
gfCNCPoint4[16490] = {X 521.3028, Y 51.1070, Z -5.5000, A 0.000, B 0.000, C 0.000 }
gfCNCPoint4[16491] = {X 520.4708, Y 51.1991, Z -5.5000, A 0.000, B 0.000, C 0.000 }
gfCNCPoint4[16492] = {X 519.7998, Y 51.1991, Z -5.5000, A 0.000, B 0.000, C 0.000 }
gfCNCPoint4[16493] = {X 518.8385, Y 51.0908, Z -5.5000, A 0.000, B 0.000, C 0.000 }
gfCNCPoint4[16494] = {X 517.9254, Y 50.7713, Z -5.5000, A 0.000, B 0.000, C 0.000 }
gfCNCPoint4[16495] = {X 517.1063, Y 50.2566, Z -5.5000, A 0.000, B 0.000, C 0.000 }
gfCNCPoint4[16496] = {X 516.4223, Y 49.5726, Z -5.5000, A 0.000, B 0.000, C 0.000 }
gfCNCPoint4[16497] = {X 515.9076, Y 48.7535, Z -5.5000, A 0.000, B 0.000, C 0.000 }
gfCNCPoint4[16498] = {X 515.5881, Y 47.8404, Z -5.5000, A 0.000, B 0.000, C 0.000 }
gfCNCPoint4[16499] = {X 515.4798, Y 46.8791, Z -5.5000, A 0.000, B 0.000, C 0.000 }
gfCNCPoint4[16500] = {X 515.4798, Y 39.9011, Z -5.5000, A 0.000, B 0.000, C 0.000 }
gfCNCPoint4[16501] = {X 515.5869, Y 38.9451, Z -5.5000, A 0.000, B 0.000, C 0.000 }
gfCNCPoint4[16502] = {X 515.9029, Y 38.0365, Z -5.5000, A 0.000, B 0.000, C 0.000 }
gfCNCPoint4[16503] = {X 516.4121, Y 37.2204, Z -5.5000, A 0.000, B 0.000, C 0.000 }
gfCNCPoint4[16504] = {X 517.0893, Y 36.5372, Z -5.5000, A 0.000, B 0.000, C 0.000 }
gfCNCPoint4[16505] = {X 517.9010, Y 36.0208, Z -5.5000, A 0.000, B 0.000, C 0.000 }
gfCNCPoint4[16506] = {X 518.8067, Y 35.6968, Z -5.5000, A 0.000, B 0.000, C 0.000 }
gfCNCPoint4[16507] = {X 519.7617, Y 35.5813, Z -5.5000, A 0.000, B 0.000, C 0.000 }
gfCNCPoint4[16508] = {X 520.5269, Y 35.5815, Z -5.5000, A 0.000, B 0.000, C 0.000 }
gfCNCPoint4[16509] = {X 521.3533, Y 35.6727, Z -5.5000, A 0.000, B 0.000, C 0.000 }
gfCNCPoint4[16510] = {X 522.1469, Y 35.9206, Z -5.5000, A 0.000, B 0.000, C 0.000 }
gfCNCPoint4[16511] = {X 522.8783, Y 36.3159, Z -5.5000, A 0.000, B 0.000, C 0.000 }
gfCNCPoint4[16512] = {X 523.5205, Y 36.8440, Z -5.5000, A 0.000, B 0.000, C 0.000 }
gfCNCPoint4[16513] = {X 524.0496, Y 37.4853, Z -5.5000, A 0.000, B 0.000, C 0.000 }
gfCNCPoint4[16514] = {X 534.6319, Y 37.4857, Z -5.5000, A 0.000, B 0.000, C 0.000 }
gfCNCPoint4[16515] = {X 534.6319, Y 33.9657, Z -5.5000, A 0.000, B 0.000, C 0.000 }
gfCNCPoint4[16516] = {X 530.1086, Y 33.9670, Z -5.5000, A 0.000, B 0.000, C 0.000 }
gfCNCPoint4[16517] = {X 529.5764, Y 34.6108, Z -5.5000, A 0.000, B 0.000, C 0.000 }
gfCNCPoint4[16518] = {X 528.9303, Y 35.1402, Z -5.5000, A 0.000, B 0.000, C 0.000 }
gfCNCPoint4[16519] = {X 528.1943, Y 35.5353, Z -5.5000, A 0.000, B 0.000, C 0.000 }
gfCNCPoint4[16520] = {X 527.3961, Y 35.7814, Z -5.5000, A 0.000, B 0.000, C 0.000 }
gfCNCPoint4[16521] = {X 526.5655, Y 35.8693, Z -5.5000, A 0.000, B 0.000, C 0.000 }
gfCNCPoint4[16522] = {X 525.8868, Y 35.8694, Z -5.5000, A 0.000, B 0.000, C 0.000 }
gfCNCPoint4[16523] = {X 524.9255, Y 35.7611, Z -5.5000, A 0.000, B 0.000, C 0.000 }
gfCNCPoint4[16524] = {X 524.0124, Y 35.4416, Z -5.5000, A 0.000, B 0.000, C 0.000 }
gfCNCPoint4[16525] = {X 523.1933, Y 34.9270, Z -5.5000, A 0.000, B 0.000, C 0.000 }
gfCNCPoint4[16526] = {X 522.5092, Y 34.2429, Z -5.5000, A 0.000, B 0.000, C 0.000 }
gfCNCPoint4[16527] = {X 521.9946, Y 33.4238, Z -5.5000, A 0.000, B 0.000, C 0.000 }
gfCNCPoint4[16528] = {X 521.6751, Y 32.5107, Z -5.5000, A 0.000, B 0.000, C 0.000 }
gfCNCPoint4[16529] = {X 521.5668, Y 31.5495, Z -5.5000, A 0.000, B 0.000, C 0.000 }
gfCNCPoint4[16530] = {X 521.5668, Y 24.5714, Z -5.5000, A 0.000, B 0.000, C 0.000 }
gfCNCPoint4[16531] = {X 521.6739, Y 23.6153, Z -5.5000, A 0.000, B 0.000, C 0.000 }
gfCNCPoint4[16532] = {X 521.9900, Y 22.7066, Z -5.5000, A 0.000, B 0.000, C 0.000 }
gfCNCPoint4[16533] = {X 522.4994, Y 21.8904, Z -5.5000, A 0.000, B 0.000, C 0.000 }
gfCNCPoint4[16534] = {X 523.1768, Y 21.2071, Z -5.5000, A 0.000, B 0.000, C 0.000 }
gfCNCPoint4[16535] = {X 523.9886, Y 20.6908, Z -5.5000, A 0.000, B 0.000, C 0.000 }
gfCNCPoint4[16536] = {X 524.8946, Y 20.3669, Z -5.5000, A 0.000, B 0.000, C 0.000 }
gfCNCPoint4[16537] = {X 525.8498, Y 20.2516, Z -5.5000, A 0.000, B 0.000, C 0.000 }
gfCNCPoint4[16538] = {X 526.5695, Y 20.2516, Z -5.5000, A 0.000, B 0.000, C 0.000 }
gfCNCPoint4[16539] = {X 527.3944, Y 20.3391, Z -5.5000, A 0.000, B 0.000, C 0.000 }
gfCNCPoint4[16540] = {X 528.1875, Y 20.5827, Z -5.5000, A 0.000, B 0.000, C 0.000 }
gfCNCPoint4[16541] = {X 528.9193, Y 20.9734, Z -5.5000, A 0.000, B 0.000, C 0.000 }
gfCNCPoint4[16542] = {X 529.5630, Y 21.4968, Z -5.5000, A 0.000, B 0.000, C 0.000 }
gfCNCPoint4[16543] = {X 530.0948, Y 22.1335, Z -5.5000, A 0.000, B 0.000, C 0.000 }
gfCNCPoint4[16544] = {X 534.6319, Y 22.1337, Z -5.5000, A 0.000, B 0.000, C 0.000 }
gfCNCPoint4[16545] = {X 534.6319, Y 19.7021, Z -5.5000, A 0.000, B 0.000, C 0.000 }
gfCNCPoint4[16546] = {X 524.1919, Y 19.7019, Z -5.5000, A 0.000, B 0.000, C 0.000 }
gfCNCPoint4[16547] = {X 523.6595, Y 20.3464, Z -5.5000, A 0.000, B 0.000, C 0.000 }
gfCNCPoint4[16548] = {X 523.0129, Y 20.8763, Z -5.5000, A 0.000, B 0.000, C 0.000 }
gfCNCPoint4[16549] = {X 522.2763, Y 21.2717, Z -5.5000, A 0.000, B 0.000, C 0.000 }
gfCNCPoint4[16550] = {X 521.4774, Y 21.5179, Z -5.5000, A 0.000, B 0.000, C 0.000 }
gfCNCPoint4[16551] = {X 520.6460, Y 21.6056, Z -5.5000, A 0.000, B 0.000, C 0.000 }
gfCNCPoint4[16552] = {X 519.9691, Y 21.6057, Z -5.5000, A 0.000, B 0.000, C 0.000 }
gfCNCPoint4[16553] = {X 519.0078, Y 21.4974, Z -5.5000, A 0.000, B 0.000, C 0.000 }
gfCNCPoint4[16554] = {X 518.0947, Y 21.1779, Z -5.5000, A 0.000, B 0.000, C 0.000 }
gfCNCPoint4[16555] = {X 517.2756, Y 20.6632, Z -5.5000, A 0.000, B 0.000, C 0.000 }
gfCNCPoint4[16556] = {X 516.5916, Y 19.9792, Z -5.5000, A 0.000, B 0.000, C 0.000 }
gfCNCPoint4[16557] = {X 516.0769, Y 19.1601, Z -5.5000, A 0.000, B 0.000, C 0.000 }
gfCNCPoint4[16558] = {X 515.7574, Y 18.2470, Z -5.5000, A 0.000, B 0.000, C 0.000 }
gfCNCPoint4[16559] = {X 515.6491, Y 17.2857, Z -5.5000, A 0.000, B 0.000, C 0.000 }
gfCNCPoint4[16560] = {X 515.6491, Y 10.3077, Z -5.5000, A 0.000, B 0.000, C 0.000 }
gfCNCPoint4[16561] = {X 515.7562, Y 9.3519, Z -5.5000, A 0.000, B 0.000, C 0.000 }
gfCNCPoint4[16562] = {X 516.0720, Y 8.4435, Z -5.5000, A 0.000, B 0.000, C 0.000 }
gfCNCPoint4[16563] = {X 516.5811, Y 7.6275, Z -5.5000, A 0.000, B 0.000, C 0.000 }
gfCNCPoint4[16564] = {X 517.2580, Y 6.9443, Z -5.5000, A 0.000, B 0.000, C 0.000 }
gfCNCPoint4[16565] = {X 518.0693, Y 6.4278, Z -5.5000, A 0.000, B 0.000, C 0.000 }
gfCNCPoint4[16566] = {X 518.9748, Y 6.1037, Z -5.5000, A 0.000, B 0.000, C 0.000 }
gfCNCPoint4[16567] = {X 519.9296, Y 5.9879, Z -5.5000, A 0.000, B 0.000, C 0.000 }
gfCNCPoint4[16568] = {X 520.6502, Y 5.9879, Z -5.5000, A 0.000, B 0.000, C 0.000 }
gfCNCPoint4[16569] = {X 521.4755, Y 6.0751, Z -5.5000, A 0.000, B 0.000, C 0.000 }
gfCNCPoint4[16570] = {X 522.2689, Y 6.3186, Z -5.5000, A 0.000, B 0.000, C 0.000 }
gfCNCPoint4[16571] = {X 523.0012, Y 6.7093, Z -5.5000, A 0.000, B 0.000, C 0.000 }
gfCNCPoint4[16572] = {X 523.6452, Y 7.2328, Z -5.5000, A 0.000, B 0.000, C 0.000 }
gfCNCPoint4[16573] = {X 524.1772, Y 7.8698, Z -5.5000, A 0.000, B 0.000, C 0.000 }
gfCNCPoint4[16574] = {X 533.9635, Y 7.8700, Z -5.5000, A 0.000, B 0.000, C 0.000 }
gfCNCPoint4[16575] = {X 533.9636, Y 3.8700, Z -5.5000, A 0.000, B 0.000, C 0.000 }
gfCNCPoint4[16576] = {X 533.9635, Y 7.9500, Z -5.5000, A 0.000, B 0.000, C 0.000 }
gfCNCPoint4[16577] = {X 543.7510, Y 7.9502, Z -5.5000, A 0.000, B 0.000, C 0.000 }
gfCNCPoint4[16578] = {X 544.7133, Y 8.0340, Z -5.5000, A 0.000, B 0.000, C 0.000 }
gfCNCPoint4[16579] = {X 545.6318, Y 8.3331, Z -5.5000, A 0.000, B 0.000, C 0.000 }
gfCNCPoint4[16580] = {X 546.4589, Y 8.8321, Z -5.5000, A 0.000, B 0.000, C 0.000 }
gfCNCPoint4[16581] = {X 547.1517, Y 9.5052, Z -5.5000, A 0.000, B 0.000, C 0.000 }
gfCNCPoint4[16582] = {X 547.6744, Y 10.3175, Z -5.5000, A 0.000, B 0.000, C 0.000 }
gfCNCPoint4[16583] = {X 547.9999, Y 11.2270, Z -5.5000, A 0.000, B 0.000, C 0.000 }
gfCNCPoint4[16584] = {X 548.1114, Y 12.1865, Z -5.5000, A 0.000, B 0.000, C 0.000 }
gfCNCPoint4[16585] = {X 548.1112, Y 13.0217, Z -5.5000, A 0.000, B 0.000, C 0.000 }
gfCNCPoint4[16586] = {X 548.0029, Y 13.9312, Z -5.5000, A 0.000, B 0.000, C 0.000 }
gfCNCPoint4[16587] = {X 547.7018, Y 14.7962, Z -5.5000, A 0.000, B 0.000, C 0.000 }
gfCNCPoint4[16588] = {X 547.2220, Y 15.5764, Z -5.5000, A 0.000, B 0.000, C 0.000 }
gfCNCPoint4[16589] = {X 546.5858, Y 16.2353, Z -5.5000, A 0.000, B 0.000, C 0.000 }
gfCNCPoint4[16590] = {X 546.5844, Y 40.9518, Z -5.5000, A 0.000, B 0.000, C 0.000 }
gfCNCPoint4[16591] = {X 546.6349, Y 40.9931, Z -5.5000, A 0.000, B 0.000, C 0.000 }
gfCNCPoint4[16592] = {X 547.2527, Y 41.6505, Z -5.5000, A 0.000, B 0.000, C 0.000 }
gfCNCPoint4[16593] = {X 547.7174, Y 42.4238, Z -5.5000, A 0.000, B 0.000, C 0.000 }
gfCNCPoint4[16594] = {X 548.0080, Y 43.2778, Z -5.5000, A 0.000, B 0.000, C 0.000 }
gfCNCPoint4[16595] = {X 548.1113, Y 44.1740, Z -5.5000, A 0.000, B 0.000, C 0.000 }
gfCNCPoint4[16596] = {X 548.1114, Y 45.0004, Z -5.5000, A 0.000, B 0.000, C 0.000 }
gfCNCPoint4[16597] = {X 548.0000, Y 45.9598, Z -5.5000, A 0.000, B 0.000, C 0.000 }
gfCNCPoint4[16598] = {X 547.6744, Y 46.8693, Z -5.5000, A 0.000, B 0.000, C 0.000 }
gfCNCPoint4[16599] = {X 547.1517, Y 47.6816, Z -5.5000, A 0.000, B 0.000, C 0.000 }
gfCNCPoint4[16600] = {X 546.4589, Y 48.3546, Z -5.5000, A 0.000, B 0.000, C 0.000 }
gfCNCPoint4[16601] = {X 545.6318, Y 48.8536, Z -5.5000, A 0.000, B 0.000, C 0.000 }
gfCNCPoint4[16602] = {X 544.7133, Y 49.1526, Z -5.5000, A 0.000, B 0.000, C 0.000 }
gfCNCPoint4[16603] = {X 543.7510, Y 49.2363, Z -5.5000, A 0.000, B 0.000, C 0.000 }
gfCNCPoint4[16604] = {X 524.0038, Y 49.2367, Z -5.5000, A 0.000, B 0.000, C 0.000 }
gfCNCPoint4[16605] = {X 523.4670, Y 49.8699, Z -5.5000, A 0.000, B 0.000, C 0.000 }
gfCNCPoint4[16606] = {X 522.8208, Y 50.3909, Z -5.5000, A 0.000, B 0.000, C 0.000 }
gfCNCPoint4[16607] = {X 522.0881, Y 50.7812, Z -5.5000, A 0.000, B 0.000, C 0.000 }
gfCNCPoint4[16608] = {X 521.2952, Y 51.0269, Z -5.5000, A 0.000, B 0.000, C 0.000 }
gfCNCPoint4[16609] = {X 520.4702, Y 51.1191, Z -5.5000, A 0.000, B 0.000, C 0.000 }
gfCNCPoint4[16610] = {X 519.7998, Y 51.1191, Z -5.5000, A 0.000, B 0.000, C 0.000 }
gfCNCPoint4[16611] = {X 518.8563, Y 51.0128, Z -5.5000, A 0.000, B 0.000, C 0.000 }
gfCNCPoint4[16612] = {X 517.9601, Y 50.6992, Z -5.5000, A 0.000, B 0.000, C 0.000 }
gfCNCPoint4[16613] = {X 517.1562, Y 50.1941, Z -5.5000, A 0.000, B 0.000, C 0.000 }
gfCNCPoint4[16614] = {X 516.4848, Y 49.5227, Z -5.5000, A 0.000, B 0.000, C 0.000 }
gfCNCPoint4[16615] = {X 515.9797, Y 48.7188, Z -5.5000, A 0.000, B 0.000, C 0.000 }
gfCNCPoint4[16616] = {X 515.6661, Y 47.8226, Z -5.5000, A 0.000, B 0.000, C 0.000 }
gfCNCPoint4[16617] = {X 515.5598, Y 46.8791, Z -5.5000, A 0.000, B 0.000, C 0.000 }
gfCNCPoint4[16618] = {X 515.5598, Y 39.9011, Z -5.5000, A 0.000, B 0.000, C 0.000 }
gfCNCPoint4[16619] = {X 515.6649, Y 38.9628, Z -5.5000, A 0.000, B 0.000, C 0.000 }
gfCNCPoint4[16620] = {X 515.9751, Y 38.0710, Z -5.5000, A 0.000, B 0.000, C 0.000 }
gfCNCPoint4[16621] = {X 516.4749, Y 37.2700, Z -5.5000, A 0.000, B 0.000, C 0.000 }
gfCNCPoint4[16622] = {X 517.1395, Y 36.5995, Z -5.5000, A 0.000, B 0.000, C 0.000 }
gfCNCPoint4[16623] = {X 517.9361, Y 36.0926, Z -5.5000, A 0.000, B 0.000, C 0.000 }
gfCNCPoint4[16624] = {X 518.8251, Y 35.7746, Z -5.5000, A 0.000, B 0.000, C 0.000 }
gfCNCPoint4[16625] = {X 519.7624, Y 35.6613, Z -5.5000, A 0.000, B 0.000, C 0.000 }
gfCNCPoint4[16626] = {X 520.5258, Y 35.6615, Z -5.5000, A 0.000, B 0.000, C 0.000 }
gfCNCPoint4[16627] = {X 521.3452, Y 35.7528, Z -5.5000, A 0.000, B 0.000, C 0.000 }
gfCNCPoint4[16628] = {X 522.1314, Y 36.0009, Z -5.5000, A 0.000, B 0.000, C 0.000 }
gfCNCPoint4[16629] = {X 522.8547, Y 36.3965, Z -5.5000, A 0.000, B 0.000, C 0.000 }
gfCNCPoint4[16630] = {X 523.4879, Y 36.9247, Z -5.5000, A 0.000, B 0.000, C 0.000 }
gfCNCPoint4[16631] = {X 524.0068, Y 37.5653, Z -5.5000, A 0.000, B 0.000, C 0.000 }
gfCNCPoint4[16632] = {X 534.7119, Y 37.5657, Z -5.5000, A 0.000, B 0.000, C 0.000 }
gfCNCPoint4[16633] = {X 534.7119, Y 33.8857, Z -5.5000, A 0.000, B 0.000, C 0.000 }
gfCNCPoint4[16634] = {X 530.0656, Y 33.8854, Z -5.5000, A 0.000, B 0.000, C 0.000 }
gfCNCPoint4[16635] = {X 530.0417, Y 33.9232, Z -5.5000, A 0.000, B 0.000, C 0.000 }
gfCNCPoint4[16636] = {X 529.5193, Y 34.5548, Z -5.5000, A 0.000, B 0.000, C 0.000 }
gfCNCPoint4[16637] = {X 528.8852, Y 35.0741, Z -5.5000, A 0.000, B 0.000, C 0.000 }
gfCNCPoint4[16638] = {X 528.1631, Y 35.4617, Z -5.5000, A 0.000, B 0.000, C 0.000 }
gfCNCPoint4[16639] = {X 527.3798, Y 35.7031, Z -5.5000, A 0.000, B 0.000, C 0.000 }
gfCNCPoint4[16640] = {X 526.5648, Y 35.7893, Z -5.5000, A 0.000, B 0.000, C 0.000 }
gfCNCPoint4[16641] = {X 525.8868, Y 35.7894, Z -5.5000, A 0.000, B 0.000, C 0.000 }
gfCNCPoint4[16642] = {X 524.9433, Y 35.6831, Z -5.5000, A 0.000, B 0.000, C 0.000 }
gfCNCPoint4[16643] = {X 524.0471, Y 35.3696, Z -5.5000, A 0.000, B 0.000, C 0.000 }
gfCNCPoint4[16644] = {X 523.2432, Y 34.8644, Z -5.5000, A 0.000, B 0.000, C 0.000 }
gfCNCPoint4[16645] = {X 522.5718, Y 34.1930, Z -5.5000, A 0.000, B 0.000, C 0.000 }
gfCNCPoint4[16646] = {X 522.0666, Y 33.3891, Z -5.5000, A 0.000, B 0.000, C 0.000 }
gfCNCPoint4[16647] = {X 521.7531, Y 32.4929, Z -5.5000, A 0.000, B 0.000, C 0.000 }
gfCNCPoint4[16648] = {X 521.6468, Y 31.5495, Z -5.5000, A 0.000, B 0.000, C 0.000 }
gfCNCPoint4[16649] = {X 521.6468, Y 24.5714, Z -5.5000, A 0.000, B 0.000, C 0.000 }
gfCNCPoint4[16650] = {X 521.7519, Y 23.6330, Z -5.5000, A 0.000, B 0.000, C 0.000 }
gfCNCPoint4[16651] = {X 522.0622, Y 22.7411, Z -5.5000, A 0.000, B 0.000, C 0.000 }
gfCNCPoint4[16652] = {X 522.5621, Y 21.9400, Z -5.5000, A 0.000, B 0.000, C 0.000 }
gfCNCPoint4[16653] = {X 523.2270, Y 21.2694, Z -5.5000, A 0.000, B 0.000, C 0.000 }
gfCNCPoint4[16654] = {X 524.0238, Y 20.7626, Z -5.5000, A 0.000, B 0.000, C 0.000 }
gfCNCPoint4[16655] = {X 524.9130, Y 20.4448, Z -5.5000, A 0.000, B 0.000, C 0.000 }
gfCNCPoint4[16656] = {X 525.8505, Y 20.3316, Z -5.5000, A 0.000, B 0.000, C 0.000 }
gfCNCPoint4[16657] = {X 526.5687, Y 20.3316, Z -5.5000, A 0.000, B 0.000, C 0.000 }
gfCNCPoint4[16658] = {X 527.3866, Y 20.4192, Z -5.5000, A 0.000, B 0.000, C 0.000 }
gfCNCPoint4[16659] = {X 528.1723, Y 20.6631, Z -5.5000, A 0.000, B 0.000, C 0.000 }
gfCNCPoint4[16660] = {X 528.8960, Y 21.0540, Z -5.5000, A 0.000, B 0.000, C 0.000 }
gfCNCPoint4[16661] = {X 529.5307, Y 21.5774, Z -5.5000, A 0.000, B 0.000, C 0.000 }
gfCNCPoint4[16662] = {X 530.0523, Y 22.2135, Z -5.5000, A 0.000, B 0.000, C 0.000 }
gfCNCPoint4[16663] = {X 534.7119, Y 22.2137, Z -5.5000, A 0.000, B 0.000, C 0.000 }
gfCNCPoint4[16664] = {X 534.7119, Y 19.6221, Z -5.5000, A 0.000, B 0.000, C 0.000 }
gfCNCPoint4[16665] = {X 524.1489, Y 19.6219, Z -5.5000, A 0.000, B 0.000, C 0.000 }
gfCNCPoint4[16666] = {X 524.1256, Y 19.6571, Z -5.5000, A 0.000, B 0.000, C 0.000 }
gfCNCPoint4[16667] = {X 523.6030, Y 20.2897, Z -5.5000, A 0.000, B 0.000, C 0.000 }
gfCNCPoint4[16668] = {X 522.9684, Y 20.8098, Z -5.5000, A 0.000, B 0.000, C 0.000 }
gfCNCPoint4[16669] = {X 522.2455, Y 21.1979, Z -5.5000, A 0.000, B 0.000, C 0.000 }
gfCNCPoint4[16670] = {X 521.4613, Y 21.4395, Z -5.5000, A 0.000, B 0.000, C 0.000 }
gfCNCPoint4[16671] = {X 520.6453, Y 21.5256, Z -5.5000, A 0.000, B 0.000, C 0.000 }
gfCNCPoint4[16672] = {X 519.9691, Y 21.5257, Z -5.5000, A 0.000, B 0.000, C 0.000 }
gfCNCPoint4[16673] = {X 519.0256, Y 21.4194, Z -5.5000, A 0.000, B 0.000, C 0.000 }
gfCNCPoint4[16674] = {X 518.1294, Y 21.1058, Z -5.5000, A 0.000, B 0.000, C 0.000 }
gfCNCPoint4[16675] = {X 517.3255, Y 20.6007, Z -5.5000, A 0.000, B 0.000, C 0.000 }
gfCNCPoint4[16676] = {X 516.6541, Y 19.9293, Z -5.5000, A 0.000, B 0.000, C 0.000 }
gfCNCPoint4[16677] = {X 516.1490, Y 19.1254, Z -5.5000, A 0.000, B 0.000, C 0.000 }
gfCNCPoint4[16678] = {X 515.8354, Y 18.2292, Z -5.5000, A 0.000, B 0.000, C 0.000 }
gfCNCPoint4[16679] = {X 515.7291, Y 17.2857, Z -5.5000, A 0.000, B 0.000, C 0.000 }
gfCNCPoint4[16680] = {X 515.7291, Y 10.3077, Z -5.5000, A 0.000, B 0.000, C 0.000 }
gfCNCPoint4[16681] = {X 515.8342, Y 9.3696, Z -5.5000, A 0.000, B 0.000, C 0.000 }
gfCNCPoint4[16682] = {X 516.1442, Y 8.4780, Z -5.5000, A 0.000, B 0.000, C 0.000 }
gfCNCPoint4[16683] = {X 516.6438, Y 7.6771, Z -5.5000, A 0.000, B 0.000, C 0.000 }
gfCNCPoint4[16684] = {X 517.3082, Y 7.0066, Z -5.5000, A 0.000, B 0.000, C 0.000 }
gfCNCPoint4[16685] = {X 518.1045, Y 6.4997, Z -5.5000, A 0.000, B 0.000, C 0.000 }
gfCNCPoint4[16686] = {X 518.9932, Y 6.1815, Z -5.5000, A 0.000, B 0.000, C 0.000 }
gfCNCPoint4[16687] = {X 519.9303, Y 6.0679, Z -5.5000, A 0.000, B 0.000, C 0.000 }
gfCNCPoint4[16688] = {X 520.6494, Y 6.0679, Z -5.5000, A 0.000, B 0.000, C 0.000 }
gfCNCPoint4[16689] = {X 521.4677, Y 6.1552, Z -5.5000, A 0.000, B 0.000, C 0.000 }
gfCNCPoint4[16690] = {X 522.2538, Y 6.3990, Z -5.5000, A 0.000, B 0.000, C 0.000 }
gfCNCPoint4[16691] = {X 522.9779, Y 6.7900, Z -5.5000, A 0.000, B 0.000, C 0.000 }
gfCNCPoint4[16692] = {X 523.6128, Y 7.3135, Z -5.5000, A 0.000, B 0.000, C 0.000 }
gfCNCPoint4[16693] = {X 524.1347, Y 7.9498, Z -5.5000, A 0.000, B 0.000, C 0.000 }
gfCNCPoint4[16694] = {X 533.9635, Y 7.9500, Z -5.5000, A 0.000, B 0.000, C 0.000 }
gfCNCPoint4[16695] = {X 533.9636, Y 3.9500, Z -5.5000, A 0.000, B 0.000, C 0.000 }
gfCNCPoint4[16696] = {X 533.9635, Y 8.0300, Z -5.5000, A 0.000, B 0.000, C 0.000 }
gfCNCPoint4[16697] = {X 543.7521, Y 8.0302, Z -5.5000, A 0.000, B 0.000, C 0.000 }
gfCNCPoint4[16698] = {X 544.6965, Y 8.1122, Z -5.5000, A 0.000, B 0.000, C 0.000 }
gfCNCPoint4[16699] = {X 545.5978, Y 8.4055, Z -5.5000, A 0.000, B 0.000, C 0.000 }
gfCNCPoint4[16700] = {X 546.4095, Y 8.8951, Z -5.5000, A 0.000, B 0.000, C 0.000 }
gfCNCPoint4[16701] = {X 547.0895, Y 9.5555, Z -5.5000, A 0.000, B 0.000, C 0.000 }
gfCNCPoint4[16702] = {X 547.6025, Y 10.3526, Z -5.5000, A 0.000, B 0.000, C 0.000 }
gfCNCPoint4[16703] = {X 547.9220, Y 11.2450, Z -5.5000, A 0.000, B 0.000, C 0.000 }
gfCNCPoint4[16704] = {X 548.0314, Y 12.1866, Z -5.5000, A 0.000, B 0.000, C 0.000 }
gfCNCPoint4[16705] = {X 548.0312, Y 13.0208, Z -5.5000, A 0.000, B 0.000, C 0.000 }
gfCNCPoint4[16706] = {X 547.9228, Y 13.9223, Z -5.5000, A 0.000, B 0.000, C 0.000 }
gfCNCPoint4[16707] = {X 547.6215, Y 14.7787, Z -5.5000, A 0.000, B 0.000, C 0.000 }
gfCNCPoint4[16708] = {X 547.1415, Y 15.5494, Z -5.5000, A 0.000, B 0.000, C 0.000 }
gfCNCPoint4[16709] = {X 546.5058, Y 16.1976, Z -5.5000, A 0.000, B 0.000, C 0.000 }
gfCNCPoint4[16710] = {X 546.5044, Y 40.9897, Z -5.5000, A 0.000, B 0.000, C 0.000 }
gfCNCPoint4[16711] = {X 546.5835, Y 41.0544, Z -5.5000, A 0.000, B 0.000, C 0.000 }
gfCNCPoint4[16712] = {X 547.1893, Y 41.6994, Z -5.5000, A 0.000, B 0.000, C 0.000 }
gfCNCPoint4[16713] = {X 547.6450, Y 42.4579, Z -5.5000, A 0.000, B 0.000, C 0.000 }
gfCNCPoint4[16714] = {X 547.9300, Y 43.2956, Z -5.5000, A 0.000, B 0.000, C 0.000 }
gfCNCPoint4[16715] = {X 548.0313, Y 44.1746, Z -5.5000, A 0.000, B 0.000, C 0.000 }
gfCNCPoint4[16716] = {X 548.0314, Y 45.0002, Z -5.5000, A 0.000, B 0.000, C 0.000 }
gfCNCPoint4[16717] = {X 547.9220, Y 45.9418, Z -5.5000, A 0.000, B 0.000, C 0.000 }
gfCNCPoint4[16718] = {X 547.6025, Y 46.8342, Z -5.5000, A 0.000, B 0.000, C 0.000 }
gfCNCPoint4[16719] = {X 547.0895, Y 47.6312, Z -5.5000, A 0.000, B 0.000, C 0.000 }
gfCNCPoint4[16720] = {X 546.4095, Y 48.2916, Z -5.5000, A 0.000, B 0.000, C 0.000 }
gfCNCPoint4[16721] = {X 545.5978, Y 48.7811, Z -5.5000, A 0.000, B 0.000, C 0.000 }
gfCNCPoint4[16722] = {X 544.6964, Y 49.0744, Z -5.5000, A 0.000, B 0.000, C 0.000 }
gfCNCPoint4[16723] = {X 543.7521, Y 49.1563, Z -5.5000, A 0.000, B 0.000, C 0.000 }
gfCNCPoint4[16724] = {X 523.9618, Y 49.1567, Z -5.5000, A 0.000, B 0.000, C 0.000 }
gfCNCPoint4[16725] = {X 523.4350, Y 49.7892, Z -5.5000, A 0.000, B 0.000, C 0.000 }
gfCNCPoint4[16726] = {X 522.7977, Y 50.3102, Z -5.5000, A 0.000, B 0.000, C 0.000 }
gfCNCPoint4[16727] = {X 522.0730, Y 50.7008, Z -5.5000, A 0.000, B 0.000, C 0.000 }
gfCNCPoint4[16728] = {X 521.2875, Y 50.9468, Z -5.5000, A 0.000, B 0.000, C 0.000 }
gfCNCPoint4[16729] = {X 520.4695, Y 51.0391, Z -5.5000, A 0.000, B 0.000, C 0.000 }
gfCNCPoint4[16730] = {X 519.7998, Y 51.0391, Z -5.5000, A 0.000, B 0.000, C 0.000 }
gfCNCPoint4[16731] = {X 518.8741, Y 50.9348, Z -5.5000, A 0.000, B 0.000, C 0.000 }
gfCNCPoint4[16732] = {X 517.9948, Y 50.6272, Z -5.5000, A 0.000, B 0.000, C 0.000 }
gfCNCPoint4[16733] = {X 517.2061, Y 50.1315, Z -5.5000, A 0.000, B 0.000, C 0.000 }
gfCNCPoint4[16734] = {X 516.5474, Y 49.4728, Z -5.5000, A 0.000, B 0.000, C 0.000 }
gfCNCPoint4[16735] = {X 516.0517, Y 48.6841, Z -5.5000, A 0.000, B 0.000, C 0.000 }
gfCNCPoint4[16736] = {X 515.7441, Y 47.8048, Z -5.5000, A 0.000, B 0.000, C 0.000 }
gfCNCPoint4[16737] = {X 515.6398, Y 46.8791, Z -5.5000, A 0.000, B 0.000, C 0.000 }
gfCNCPoint4[16738] = {X 515.6398, Y 39.9011, Z -5.5000, A 0.000, B 0.000, C 0.000 }
gfCNCPoint4[16739] = {X 515.7429, Y 38.9805, Z -5.5000, A 0.000, B 0.000, C 0.000 }
gfCNCPoint4[16740] = {X 516.0472, Y 38.1056, Z -5.5000, A 0.000, B 0.000, C 0.000 }
gfCNCPoint4[16741] = {X 516.5376, Y 37.3197, Z -5.5000, A 0.000, B 0.000, C 0.000 }
gfCNCPoint4[16742] = {X 517.1897, Y 36.6618, Z -5.5000, A 0.000, B 0.000, C 0.000 }
gfCNCPoint4[16743] = {X 517.9713, Y 36.1645, Z -5.5000, A 0.000, B 0.000, C 0.000 }
gfCNCPoint4[16744] = {X 518.8435, Y 35.8525, Z -5.5000, A 0.000, B 0.000, C 0.000 }
gfCNCPoint4[16745] = {X 519.7631, Y 35.7413, Z -5.5000, A 0.000, B 0.000, C 0.000 }
gfCNCPoint4[16746] = {X 520.5247, Y 35.7415, Z -5.5000, A 0.000, B 0.000, C 0.000 }
gfCNCPoint4[16747] = {X 521.3370, Y 35.8328, Z -5.5000, A 0.000, B 0.000, C 0.000 }
gfCNCPoint4[16748] = {X 522.1158, Y 36.0813, Z -5.5000, A 0.000, B 0.000, C 0.000 }
gfCNCPoint4[16749] = {X 522.8309, Y 36.4772, Z -5.5000, A 0.000, B 0.000, C 0.000 }
gfCNCPoint4[16750] = {X 523.4549, Y 37.0054, Z -5.5000, A 0.000, B 0.000, C 0.000 }
gfCNCPoint4[16751] = {X 523.9635, Y 37.6453, Z -5.5000, A 0.000, B 0.000, C 0.000 }
gfCNCPoint4[16752] = {X 534.7919, Y 37.6457, Z -5.5000, A 0.000, B 0.000, C 0.000 }
gfCNCPoint4[16753] = {X 534.7919, Y 33.8057, Z -5.5000, A 0.000, B 0.000, C 0.000 }
gfCNCPoint4[16754] = {X 530.0216, Y 33.8054, Z -5.5000, A 0.000, B 0.000, C 0.000 }
gfCNCPoint4[16755] = {X 529.9747, Y 33.8794, Z -5.5000, A 0.000, B 0.000, C 0.000 }
gfCNCPoint4[16756] = {X 529.4622, Y 34.4988, Z -5.5000, A 0.000, B 0.000, C 0.000 }
gfCNCPoint4[16757] = {X 528.8402, Y 35.0080, Z -5.5000, A 0.000, B 0.000, C 0.000 }
gfCNCPoint4[16758] = {X 528.1318, Y 35.3881, Z -5.5000, A 0.000, B 0.000, C 0.000 }
gfCNCPoint4[16759] = {X 527.3635, Y 35.6248, Z -5.5000, A 0.000, B 0.000, C 0.000 }
gfCNCPoint4[16760] = {X 526.5641, Y 35.7093, Z -5.5000, A 0.000, B 0.000, C 0.000 }
gfCNCPoint4[16761] = {X 525.8868, Y 35.7094, Z -5.5000, A 0.000, B 0.000, C 0.000 }
gfCNCPoint4[16762] = {X 524.9611, Y 35.6051, Z -5.5000, A 0.000, B 0.000, C 0.000 }
gfCNCPoint4[16763] = {X 524.0818, Y 35.2975, Z -5.5000, A 0.000, B 0.000, C 0.000 }
gfCNCPoint4[16764] = {X 523.2930, Y 34.8019, Z -5.5000, A 0.000, B 0.000, C 0.000 }
gfCNCPoint4[16765] = {X 522.6343, Y 34.1432, Z -5.5000, A 0.000, B 0.000, C 0.000 }
gfCNCPoint4[16766] = {X 522.1387, Y 33.3544, Z -5.5000, A 0.000, B 0.000, C 0.000 }
gfCNCPoint4[16767] = {X 521.8311, Y 32.4751, Z -5.5000, A 0.000, B 0.000, C 0.000 }
gfCNCPoint4[16768] = {X 521.7268, Y 31.5495, Z -5.5000, A 0.000, B 0.000, C 0.000 }
gfCNCPoint4[16769] = {X 521.7268, Y 24.5714, Z -5.5000, A 0.000, B 0.000, C 0.000 }
gfCNCPoint4[16770] = {X 521.8299, Y 23.6507, Z -5.5000, A 0.000, B 0.000, C 0.000 }
gfCNCPoint4[16771] = {X 522.1343, Y 22.7756, Z -5.5000, A 0.000, B 0.000, C 0.000 }
gfCNCPoint4[16772] = {X 522.6248, Y 21.9897, Z -5.5000, A 0.000, B 0.000, C 0.000 }
gfCNCPoint4[16773] = {X 523.2772, Y 21.3317, Z -5.5000, A 0.000, B 0.000, C 0.000 }
gfCNCPoint4[16774] = {X 524.0589, Y 20.8345, Z -5.5000, A 0.000, B 0.000, C 0.000 }
gfCNCPoint4[16775] = {X 524.9313, Y 20.5226, Z -5.5000, A 0.000, B 0.000, C 0.000 }
gfCNCPoint4[16776] = {X 525.8511, Y 20.4116, Z -5.5000, A 0.000, B 0.000, C 0.000 }
gfCNCPoint4[16777] = {X 526.5679, Y 20.4116, Z -5.5000, A 0.000, B 0.000, C 0.000 }
gfCNCPoint4[16778] = {X 527.3788, Y 20.4993, Z -5.5000, A 0.000, B 0.000, C 0.000 }
gfCNCPoint4[16779] = {X 528.1570, Y 20.7434, Z -5.5000, A 0.000, B 0.000, C 0.000 }
gfCNCPoint4[16780] = {X 528.8725, Y 21.1347, Z -5.5000, A 0.000, B 0.000, C 0.000 }
gfCNCPoint4[16781] = {X 529.4980, Y 21.6581, Z -5.5000, A 0.000, B 0.000, C 0.000 }
gfCNCPoint4[16782] = {X 530.0093, Y 22.2935, Z -5.5000, A 0.000, B 0.000, C 0.000 }
gfCNCPoint4[16783] = {X 534.7919, Y 22.2937, Z -5.5000, A 0.000, B 0.000, C 0.000 }
gfCNCPoint4[16784] = {X 534.7919, Y 19.5421, Z -5.5000, A 0.000, B 0.000, C 0.000 }
gfCNCPoint4[16785] = {X 524.1049, Y 19.5419, Z -5.5000, A 0.000, B 0.000, C 0.000 }
gfCNCPoint4[16786] = {X 524.0762, Y 19.5871, Z -5.5000, A 0.000, B 0.000, C 0.000 }
gfCNCPoint4[16787] = {X 523.5638, Y 20.2158, Z -5.5000, A 0.000, B 0.000, C 0.000 }
gfCNCPoint4[16788] = {X 522.9391, Y 20.7331, Z -5.5000, A 0.000, B 0.000, C 0.000 }
gfCNCPoint4[16789] = {X 522.2259, Y 21.1194, Z -5.5000, A 0.000, B 0.000, C 0.000 }
gfCNCPoint4[16790] = {X 521.4512, Y 21.3599, Z -5.5000, A 0.000, B 0.000, C 0.000 }
gfCNCPoint4[16791] = {X 520.6447, Y 21.4456, Z -5.5000, A 0.000, B 0.000, C 0.000 }
gfCNCPoint4[16792] = {X 519.9691, Y 21.4457, Z -5.5000, A 0.000, B 0.000, C 0.000 }
gfCNCPoint4[16793] = {X 519.0434, Y 21.3414, Z -5.5000, A 0.000, B 0.000, C 0.000 }
gfCNCPoint4[16794] = {X 518.1641, Y 21.0337, Z -5.5000, A 0.000, B 0.000, C 0.000 }
gfCNCPoint4[16795] = {X 517.3754, Y 20.5381, Z -5.5000, A 0.000, B 0.000, C 0.000 }
gfCNCPoint4[16796] = {X 516.7167, Y 19.8794, Z -5.5000, A 0.000, B 0.000, C 0.000 }
gfCNCPoint4[16797] = {X 516.2211, Y 19.0907, Z -5.5000, A 0.000, B 0.000, C 0.000 }
gfCNCPoint4[16798] = {X 515.9134, Y 18.2114, Z -5.5000, A 0.000, B 0.000, C 0.000 }
gfCNCPoint4[16799] = {X 515.8091, Y 17.2857, Z -5.5000, A 0.000, B 0.000, C 0.000 }
gfCNCPoint4[16800] = {X 515.8091, Y 10.3077, Z -5.5000, A 0.000, B 0.000, C 0.000 }
gfCNCPoint4[16801] = {X 515.9122, Y 9.3873, Z -5.5000, A 0.000, B 0.000, C 0.000 }
gfCNCPoint4[16802] = {X 516.2164, Y 8.5125, Z -5.5000, A 0.000, B 0.000, C 0.000 }
gfCNCPoint4[16803] = {X 516.7065, Y 7.7267, Z -5.5000, A 0.000, B 0.000, C 0.000 }
gfCNCPoint4[16804] = {X 517.3584, Y 7.0689, Z -5.5000, A 0.000, B 0.000, C 0.000 }
gfCNCPoint4[16805] = {X 518.1397, Y 6.5715, Z -5.5000, A 0.000, B 0.000, C 0.000 }
gfCNCPoint4[16806] = {X 519.0117, Y 6.2594, Z -5.5000, A 0.000, B 0.000, C 0.000 }
gfCNCPoint4[16807] = {X 519.9311, Y 6.1479, Z -5.5000, A 0.000, B 0.000, C 0.000 }
gfCNCPoint4[16808] = {X 520.6487, Y 6.1479, Z -5.5000, A 0.000, B 0.000, C 0.000 }
gfCNCPoint4[16809] = {X 521.4599, Y 6.2353, Z -5.5000, A 0.000, B 0.000, C 0.000 }
gfCNCPoint4[16810] = {X 522.2384, Y 6.4793, Z -5.5000, A 0.000, B 0.000, C 0.000 }
gfCNCPoint4[16811] = {X 522.9544, Y 6.8707, Z -5.5000, A 0.000, B 0.000, C 0.000 }
gfCNCPoint4[16812] = {X 523.5802, Y 7.3942, Z -5.5000, A 0.000, B 0.000, C 0.000 }
gfCNCPoint4[16813] = {X 524.0917, Y 8.0298, Z -5.5000, A 0.000, B 0.000, C 0.000 }
gfCNCPoint4[16814] = {X 533.9635, Y 8.0300, Z -5.5000, A 0.000, B 0.000, C 0.000 }
gfCNCPoint4[16815] = {X 533.9636, Y 4.0300, Z -5.5000, A 0.000, B 0.000, C 0.000 }
gfCNCPoint4[16816] = {X 533.9635, Y 8.1100, Z -5.5000, A 0.000, B 0.000, C 0.000 }
gfCNCPoint4[16817] = {X 543.7532, Y 8.1102, Z -5.5000, A 0.000, B 0.000, C 0.000 }
gfCNCPoint4[16818] = {X 544.6796, Y 8.1904, Z -5.5000, A 0.000, B 0.000, C 0.000 }
gfCNCPoint4[16819] = {X 545.5639, Y 8.4780, Z -5.5000, A 0.000, B 0.000, C 0.000 }
gfCNCPoint4[16820] = {X 546.3602, Y 8.9581, Z -5.5000, A 0.000, B 0.000, C 0.000 }
gfCNCPoint4[16821] = {X 547.0273, Y 9.6058, Z -5.5000, A 0.000, B 0.000, C 0.000 }
gfCNCPoint4[16822] = {X 547.5306, Y 10.3877, Z -5.5000, A 0.000, B 0.000, C 0.000 }
gfCNCPoint4[16823] = {X 547.8441, Y 11.2631, Z -5.5000, A 0.000, B 0.000, C 0.000 }
gfCNCPoint4[16824] = {X 547.9514, Y 12.1867, Z -5.5000, A 0.000, B 0.000, C 0.000 }
gfCNCPoint4[16825] = {X 547.9512, Y 13.0200, Z -5.5000, A 0.000, B 0.000, C 0.000 }
gfCNCPoint4[16826] = {X 547.8428, Y 13.9133, Z -5.5000, A 0.000, B 0.000, C 0.000 }
gfCNCPoint4[16827] = {X 547.5412, Y 14.7611, Z -5.5000, A 0.000, B 0.000, C 0.000 }
gfCNCPoint4[16828] = {X 547.0611, Y 15.5222, Z -5.5000, A 0.000, B 0.000, C 0.000 }
gfCNCPoint4[16829] = {X 546.4258, Y 16.1595, Z -5.5000, A 0.000, B 0.000, C 0.000 }
gfCNCPoint4[16830] = {X 546.4244, Y 41.0277, Z -5.5000, A 0.000, B 0.000, C 0.000 }
gfCNCPoint4[16831] = {X 546.5322, Y 41.1157, Z -5.5000, A 0.000, B 0.000, C 0.000 }
gfCNCPoint4[16832] = {X 547.1260, Y 41.7482, Z -5.5000, A 0.000, B 0.000, C 0.000 }
gfCNCPoint4[16833] = {X 547.5727, Y 42.4920, Z -5.5000, A 0.000, B 0.000, C 0.000 }
gfCNCPoint4[16834] = {X 547.8520, Y 43.3134, Z -5.5000, A 0.000, B 0.000, C 0.000 }
gfCNCPoint4[16835] = {X 547.9513, Y 44.1753, Z -5.5000, A 0.000, B 0.000, C 0.000 }
gfCNCPoint4[16836] = {X 547.9514, Y 45.0001, Z -5.5000, A 0.000, B 0.000, C 0.000 }
gfCNCPoint4[16837] = {X 547.8441, Y 45.9237, Z -5.5000, A 0.000, B 0.000, C 0.000 }
gfCNCPoint4[16838] = {X 547.5306, Y 46.7991, Z -5.5000, A 0.000, B 0.000, C 0.000 }
gfCNCPoint4[16839] = {X 547.0273, Y 47.5809, Z -5.5000, A 0.000, B 0.000, C 0.000 }
gfCNCPoint4[16840] = {X 546.3602, Y 48.2287, Z -5.5000, A 0.000, B 0.000, C 0.000 }
gfCNCPoint4[16841] = {X 545.5639, Y 48.7087, Z -5.5000, A 0.000, B 0.000, C 0.000 }
gfCNCPoint4[16842] = {X 544.6796, Y 48.9962, Z -5.5000, A 0.000, B 0.000, C 0.000 }
gfCNCPoint4[16843] = {X 543.7532, Y 49.0763, Z -5.5000, A 0.000, B 0.000, C 0.000 }
